gfCNCPoint4[9687] = {X 25.0315, Y 46.1433, Z -5.5000, A 0.000, B 0.000, C 0.000 }
gfCNCPoint4[9688] = {X 23.2598, Y 47.0763, Z -5.5000, A 0.000, B 0.000, C 0.000 }
gfCNCPoint4[9689] = {X 21.4277, Y 47.8844, Z -5.5000, A 0.000, B 0.000, C 0.000 }
gfCNCPoint4[9690] = {X 19.5440, Y 48.5635, Z -5.5000, A 0.000, B 0.000, C 0.000 }
gfCNCPoint4[9691] = {X 19.3880, Y 48.6154, Z -5.5000, A 0.000, B 0.000, C 0.000 }
gfCNCPoint4[9692] = {X 17.4978, Y 49.1350, Z -5.5000, A 0.000, B 0.000, C 0.000 }
gfCNCPoint4[9693] = {X 15.5694, Y 49.4877, Z -5.5000, A 0.000, B 0.000, C 0.000 }
gfCNCPoint4[9694] = {X 13.6177, Y 49.6708, Z -5.5000, A 0.000, B 0.000, C 0.000 }
gfCNCPoint4[9695] = {X 11.6574, Y 49.6828, Z -5.5000, A 0.000, B 0.000, C 0.000 }
gfCNCPoint4[9696] = {X 9.7035, Y 49.5238, Z -5.5000, A 0.000, B 0.000, C 0.000 }
gfCNCPoint4[9697] = {X 7.7709, Y 49.1949, Z -5.5000, A 0.000, B 0.000, C 0.000 }
gfCNCPoint4[9698] = {X 5.9054, Y 48.6841, Z -5.5000, A 0.000, B 0.000, C 0.000 }
gfCNCPoint4[9699] = {X 4.1131, Y 47.9568, Z -5.5000, A 0.000, B 0.000, C 0.000 }
gfCNCPoint4[9700] = {X 2.4191, Y 47.0233, Z -5.5000, A 0.000, B 0.000, C 0.000 }
gfCNCPoint4[9701] = {X 0.8469, Y 45.8966, Z -5.5000, A 0.000, B 0.000, C 0.000 }
gfCNCPoint4[9702] = {X -0.2578, Y 44.9037, Z -5.5000, A 0.000, B 0.000, C 0.000 }
gfCNCPoint4[9703] = {X -1.2389, Y 43.7885, Z -5.5000, A 0.000, B 0.000, C 0.000 }
gfCNCPoint4[9704] = {X -2.0830, Y 42.5663, Z -5.5000, A 0.000, B 0.000, C 0.000 }
gfCNCPoint4[9705] = {X -2.7785, Y 41.2539, Z -5.5000, A 0.000, B 0.000, C 0.000 }
gfCNCPoint4[9706] = {X -3.3159, Y 39.8692, Z -5.5000, A 0.000, B 0.000, C 0.000 }
gfCNCPoint4[9707] = {X -3.5286, Y 39.1333, Z -5.5000, A 0.000, B 0.000, C 0.000 }
gfCNCPoint4[9708] = {X -3.6966, Y 38.3859, Z -5.5000, A 0.000, B 0.000, C 0.000 }
gfCNCPoint4[9709] = {X -4.4555, Y 34.4585, Z -5.5000, A 0.000, B 0.000, C 0.000 }
gfCNCPoint4[9710] = {X -7.9739, Y 34.2502, Z -5.5000, A 0.000, B 0.000, C 0.000 }
gfCNCPoint4[9711] = {X -7.9739, Y 34.2502, Z -2.5000, A 0.000, B 0.000, C 0.000 }
gfCNCPoint4[9712] = {X -7.9739, Y 34.2502, Z 11.0000, A 0.000, B 0.000, C 0.000 }
gfCNCPoint4[9713] = {X 39.8247, Y 26.3830, Z 11.0000, A 0.000, B 0.000, C 0.000 }
gfCNCPoint4[9714] = {X 39.8247, Y 26.3830, Z -2.5000, A 0.000, B 0.000, C 0.000 }
gfCNCPoint4[9715] = {X 39.8247, Y 26.3830, Z -5.5000, A 0.000, B 0.000, C 0.000 }
gfCNCPoint4[9716] = {X 43.6481, Y 27.8072, Z -5.5000, A 0.000, B 0.000, C 0.000 }
gfCNCPoint4[9717] = {X 48.2901, Y 15.3446, Z -5.5000, A 0.000, B 0.000, C 0.000 }
gfCNCPoint4[9718] = {X 47.9079, Y 14.6186, Z -5.5000, A 0.000, B 0.000, C 0.000 }
gfCNCPoint4[9719] = {X 47.6698, Y 13.8334, Z -5.5000, A 0.000, B 0.000, C 0.000 }
gfCNCPoint4[9720] = {X 47.5844, Y 13.0173, Z -5.5000, A 0.000, B 0.000, C 0.000 }
gfCNCPoint4[9721] = {X 47.5842, Y 12.1868, Z -5.5000, A 0.000, B 0.000, C 0.000 }
gfCNCPoint4[9722] = {X 47.6925, Y 11.2255, Z -5.5000, A 0.000, B 0.000, C 0.000 }
gfCNCPoint4[9723] = {X 48.0120, Y 10.3125, Z -5.5000, A 0.000, B 0.000, C 0.000 }
gfCNCPoint4[9724] = {X 48.5267, Y 9.4933, Z -5.5000, A 0.000, B 0.000, C 0.000 }
gfCNCPoint4[9725] = {X 49.2107, Y 8.8093, Z -5.5000, A 0.000, B 0.000, C 0.000 }
gfCNCPoint4[9726] = {X 50.0298, Y 8.2946, Z -5.5000, A 0.000, B 0.000, C 0.000 }
gfCNCPoint4[9727] = {X 50.9429, Y 7.9751, Z -5.5000, A 0.000, B 0.000, C 0.000 }
gfCNCPoint4[9728] = {X 51.9042, Y 7.8668, Z -5.5000, A 0.000, B 0.000, C 0.000 }
gfCNCPoint4[9729] = {X 59.6221, Y 7.8668, Z -5.5000, A 0.000, B 0.000, C 0.000 }
gfCNCPoint4[9730] = {X 60.5834, Y 7.9751, Z -5.5000, A 0.000, B 0.000, C 0.000 }
gfCNCPoint4[9731] = {X 61.4965, Y 8.2946, Z -5.5000, A 0.000, B 0.000, C 0.000 }
gfCNCPoint4[9732] = {X 62.3156, Y 8.8093, Z -5.5000, A 0.000, B 0.000, C 0.000 }
gfCNCPoint4[9733] = {X 62.9996, Y 9.4933, Z -5.5000, A 0.000, B 0.000, C 0.000 }
gfCNCPoint4[9734] = {X 63.5143, Y 10.3124, Z -5.5000, A 0.000, B 0.000, C 0.000 }
gfCNCPoint4[9735] = {X 63.8338, Y 11.2255, Z -5.5000, A 0.000, B 0.000, C 0.000 }
gfCNCPoint4[9736] = {X 63.9421, Y 12.1868, Z -5.5000, A 0.000, B 0.000, C 0.000 }
gfCNCPoint4[9737] = {X 63.9421, Y 12.9782, Z -5.5000, A 0.000, B 0.000, C 0.000 }
gfCNCPoint4[9738] = {X 63.8584, Y 13.8245, Z -5.5000, A 0.000, B 0.000, C 0.000 }
gfCNCPoint4[9739] = {X 63.6104, Y 14.6381, Z -5.5000, A 0.000, B 0.000, C 0.000 }
gfCNCPoint4[9740] = {X 63.2079, Y 15.3874, Z -5.5000, A 0.000, B 0.000, C 0.000 }
gfCNCPoint4[9741] = {X 63.4261, Y 15.9633, Z -5.5000, A 0.000, B 0.000, C 0.000 }
gfCNCPoint4[9742] = {X 66.2401, Y 23.4308, Z -5.5000, A 0.000, B 0.000, C 0.000 }
gfCNCPoint4[9743] = {X 72.2100, Y 39.5004, Z -5.5000, A 0.000, B 0.000, C 0.000 }
gfCNCPoint4[9744] = {X 72.5154, Y 40.2685, Z -5.5000, A 0.000, B 0.000, C 0.000 }
gfCNCPoint4[9745] = {X 73.3597, Y 40.7703, Z -5.5000, A 0.000, B 0.000, C 0.000 }
gfCNCPoint4[9746] = {X 74.0688, Y 41.4499, Z -5.5000, A 0.000, B 0.000, C 0.000 }
gfCNCPoint4[9747] = {X 74.6060, Y 42.2721, Z -5.5000, A 0.000, B 0.000, C 0.000 }
gfCNCPoint4[9748] = {X 74.9437, Y 43.1944, Z -5.5000, A 0.000, B 0.000, C 0.000 }
gfCNCPoint4[9749] = {X 75.0643, Y 44.1692, Z -5.5000, A 0.000, B 0.000, C 0.000 }
gfCNCPoint4[9750] = {X 75.0645, Y 45.0000, Z -5.5000, A 0.000, B 0.000, C 0.000 }
gfCNCPoint4[9751] = {X 74.9561, Y 45.9613, Z -5.5000, A 0.000, B 0.000, C 0.000 }
gfCNCPoint4[9752] = {X 74.6366, Y 46.8744, Z -5.5000, A 0.000, B 0.000, C 0.000 }
gfCNCPoint4[9753] = {X 74.1220, Y 47.6935, Z -5.5000, A 0.000, B 0.000, C 0.000 }
gfCNCPoint4[9754] = {X 73.4379, Y 48.3775, Z -5.5000, A 0.000, B 0.000, C 0.000 }
gfCNCPoint4[9755] = {X 72.6188, Y 48.8922, Z -5.5000, A 0.000, B 0.000, C 0.000 }
gfCNCPoint4[9756] = {X 71.7057, Y 49.2117, Z -5.5000, A 0.000, B 0.000, C 0.000 }
gfCNCPoint4[9757] = {X 70.7445, Y 49.3200, Z -5.5000, A 0.000, B 0.000, C 0.000 }
gfCNCPoint4[9758] = {X 64.1851, Y 49.3200, Z -5.5000, A 0.000, B 0.000, C 0.000 }
gfCNCPoint4[9759] = {X 63.2238, Y 49.2117, Z -5.5000, A 0.000, B 0.000, C 0.000 }
gfCNCPoint4[9760] = {X 62.3108, Y 48.8922, Z -5.5000, A 0.000, B 0.000, C 0.000 }
gfCNCPoint4[9761] = {X 61.4917, Y 48.3775, Z -5.5000, A 0.000, B 0.000, C 0.000 }
gfCNCPoint4[9762] = {X 60.8076, Y 47.6935, Z -5.5000, A 0.000, B 0.000, C 0.000 }
gfCNCPoint4[9763] = {X 60.2929, Y 46.8744, Z -5.5000, A 0.000, B 0.000, C 0.000 }
gfCNCPoint4[9764] = {X 59.9734, Y 45.9613, Z -5.5000, A 0.000, B 0.000, C 0.000 }
gfCNCPoint4[9765] = {X 59.8651, Y 45.0000, Z -5.5000, A 0.000, B 0.000, C 0.000 }
gfCNCPoint4[9766] = {X 59.8651, Y 44.2085, Z -5.5000, A 0.000, B 0.000, C 0.000 }
gfCNCPoint4[9767] = {X 59.9518, Y 43.3502, Z -5.5000, A 0.000, B 0.000, C 0.000 }
gfCNCPoint4[9768] = {X 60.2072, Y 42.5262, Z -5.5000, A 0.000, B 0.000, C 0.000 }
gfCNCPoint4[9769] = {X 60.6213, Y 41.7694, Z -5.5000, A 0.000, B 0.000, C 0.000 }
gfCNCPoint4[9770] = {X 60.0068, Y 40.0892, Z -5.5000, A 0.000, B 0.000, C 0.000 }
gfCNCPoint4[9771] = {X 52.0776, Y 40.0892, Z -5.5000, A 0.000, B 0.000, C 0.000 }
gfCNCPoint4[9772] = {X 51.3347, Y 42.0851, Z -5.5000, A 0.000, B 0.000, C 0.000 }
gfCNCPoint4[9773] = {X 51.3378, Y 42.0902, Z -5.5000, A 0.000, B 0.000, C 0.000 }
gfCNCPoint4[9774] = {X 51.6390, Y 42.7496, Z -5.5000, A 0.000, B 0.000, C 0.000 }
gfCNCPoint4[9775] = {X 51.8258, Y 43.4501, Z -5.5000, A 0.000, B 0.000, C 0.000 }
gfCNCPoint4[9776] = {X 51.8928, Y 44.1720, Z -5.5000, A 0.000, B 0.000, C 0.000 }
gfCNCPoint4[9777] = {X 51.8929, Y 45.0000, Z -5.5000, A 0.000, B 0.000, C 0.000 }
gfCNCPoint4[9778] = {X 51.7846, Y 45.9613, Z -5.5000, A 0.000, B 0.000, C 0.000 }
gfCNCPoint4[9779] = {X 51.4651, Y 46.8744, Z -5.5000, A 0.000, B 0.000, C 0.000 }
gfCNCPoint4[9780] = {X 50.9504, Y 47.6935, Z -5.5000, A 0.000, B 0.000, C 0.000 }
gfCNCPoint4[9781] = {X 50.2664, Y 48.3775, Z -5.5000, A 0.000, B 0.000, C 0.000 }
gfCNCPoint4[9782] = {X 49.4473, Y 48.8922, Z -5.5000, A 0.000, B 0.000, C 0.000 }
gfCNCPoint4[9783] = {X 48.5342, Y 49.2117, Z -5.5000, A 0.000, B 0.000, C 0.000 }
gfCNCPoint4[9784] = {X 47.5729, Y 49.3200, Z -5.5000, A 0.000, B 0.000, C 0.000 }
gfCNCPoint4[9785] = {X 40.6393, Y 49.3200, Z -5.5000, A 0.000, B 0.000, C 0.000 }
gfCNCPoint4[9786] = {X 39.6780, Y 49.2117, Z -5.5000, A 0.000, B 0.000, C 0.000 }
gfCNCPoint4[9787] = {X 38.7649, Y 48.8922, Z -5.5000, A 0.000, B 0.000, C 0.000 }
gfCNCPoint4[9788] = {X 37.9458, Y 48.3775, Z -5.5000, A 0.000, B 0.000, C 0.000 }
gfCNCPoint4[9789] = {X 37.2618, Y 47.6935, Z -5.5000, A 0.000, B 0.000, C 0.000 }
gfCNCPoint4[9790] = {X 36.7471, Y 46.8744, Z -5.5000, A 0.000, B 0.000, C 0.000 }
gfCNCPoint4[9791] = {X 36.4276, Y 45.9613, Z -5.5000, A 0.000, B 0.000, C 0.000 }
gfCNCPoint4[9792] = {X 36.3193, Y 45.0000, Z -5.5000, A 0.000, B 0.000, C 0.000 }
gfCNCPoint4[9793] = {X 36.3193, Y 44.2086, Z -5.5000, A 0.000, B 0.000, C 0.000 }
gfCNCPoint4[9794] = {X 36.4360, Y 43.2115, Z -5.5000, A 0.000, B 0.000, C 0.000 }
gfCNCPoint4[9795] = {X 36.7796, Y 42.2683, Z -5.5000, A 0.000, B 0.000, C 0.000 }
gfCNCPoint4[9796] = {X 37.3317, Y 41.4299, Z -5.5000, A 0.000, B 0.000, C 0.000 }
gfCNCPoint4[9797] = {X 38.0624, Y 40.7415, Z -5.5000, A 0.000, B 0.000, C 0.000 }
gfCNCPoint4[9798] = {X 38.9322, Y 40.2404, Z -5.5000, A 0.000, B 0.000, C 0.000 }
gfCNCPoint4[9799] = {X 39.5233, Y 38.8448, Z -5.5000, A 0.000, B 0.000, C 0.000 }
gfCNCPoint4[9800] = {X 40.0641, Y 37.4291, Z -5.5000, A 0.000, B 0.000, C 0.000 }
gfCNCPoint4[9801] = {X 43.6481, Y 27.8072, Z -5.5000, A 0.000, B 0.000, C 0.000 }
gfCNCPoint4[9802] = {X 39.8997, Y 26.4110, Z -5.5000, A 0.000, B 0.000, C 0.000 }
gfCNCPoint4[9803] = {X 43.7231, Y 27.8351, Z -5.5000, A 0.000, B 0.000, C 0.000 }
gfCNCPoint4[9804] = {X 48.3793, Y 15.3344, Z -5.5000, A 0.000, B 0.000, C 0.000 }
gfCNCPoint4[9805] = {X 47.9922, Y 14.6130, Z -5.5000, A 0.000, B 0.000, C 0.000 }
gfCNCPoint4[9806] = {X 47.7508, Y 13.8307, Z -5.5000, A 0.000, B 0.000, C 0.000 }
gfCNCPoint4[9807] = {X 47.6644, Y 13.0166, Z -5.5000, A 0.000, B 0.000, C 0.000 }
gfCNCPoint4[9808] = {X 47.6642, Y 12.1868, Z -5.5000, A 0.000, B 0.000, C 0.000 }
gfCNCPoint4[9809] = {X 47.7705, Y 11.2433, Z -5.5000, A 0.000, B 0.000, C 0.000 }
gfCNCPoint4[9810] = {X 48.0841, Y 10.3472, Z -5.5000, A 0.000, B 0.000, C 0.000 }
gfCNCPoint4[9811] = {X 48.5893, Y 9.5432, Z -5.5000, A 0.000, B 0.000, C 0.000 }
gfCNCPoint4[9812] = {X 49.2606, Y 8.8719, Z -5.5000, A 0.000, B 0.000, C 0.000 }
gfCNCPoint4[9813] = {X 50.0646, Y 8.3667, Z -5.5000, A 0.000, B 0.000, C 0.000 }
gfCNCPoint4[9814] = {X 50.9607, Y 8.0531, Z -5.5000, A 0.000, B 0.000, C 0.000 }
gfCNCPoint4[9815] = {X 51.9042, Y 7.9468, Z -5.5000, A 0.000, B 0.000, C 0.000 }
gfCNCPoint4[9816] = {X 59.6221, Y 7.9468, Z -5.5000, A 0.000, B 0.000, C 0.000 }
gfCNCPoint4[9817] = {X 60.5656, Y 8.0531, Z -5.5000, A 0.000, B 0.000, C 0.000 }
gfCNCPoint4[9818] = {X 61.4618, Y 8.3667, Z -5.5000, A 0.000, B 0.000, C 0.000 }
gfCNCPoint4[9819] = {X 62.2657, Y 8.8718, Z -5.5000, A 0.000, B 0.000, C 0.000 }
gfCNCPoint4[9820] = {X 62.9371, Y 9.5432, Z -5.5000, A 0.000, B 0.000, C 0.000 }
gfCNCPoint4[9821] = {X 63.4422, Y 10.3471, Z -5.5000, A 0.000, B 0.000, C 0.000 }
gfCNCPoint4[9822] = {X 63.7558, Y 11.2433, Z -5.5000, A 0.000, B 0.000, C 0.000 }
gfCNCPoint4[9823] = {X 63.8621, Y 12.1868, Z -5.5000, A 0.000, B 0.000, C 0.000 }
gfCNCPoint4[9824] = {X 63.8621, Y 12.9782, Z -5.5000, A 0.000, B 0.000, C 0.000 }
gfCNCPoint4[9825] = {X 63.7772, Y 13.8223, Z -5.5000, A 0.000, B 0.000, C 0.000 }
gfCNCPoint4[9826] = {X 63.5259, Y 14.6327, Z -5.5000, A 0.000, B 0.000, C 0.000 }
gfCNCPoint4[9827] = {X 63.1183, Y 15.3768, Z -5.5000, A 0.000, B 0.000, C 0.000 }
gfCNCPoint4[9828] = {X 63.3513, Y 15.9916, Z -5.5000, A 0.000, B 0.000, C 0.000 }
gfCNCPoint4[9829] = {X 66.1652, Y 23.4588, Z -5.5000, A 0.000, B 0.000, C 0.000 }
gfCNCPoint4[9830] = {X 72.1353, Y 39.5291, Z -5.5000, A 0.000, B 0.000, C 0.000 }
gfCNCPoint4[9831] = {X 72.4531, Y 40.3283, Z -5.5000, A 0.000, B 0.000, C 0.000 }
gfCNCPoint4[9832] = {X 73.2906, Y 40.8184, Z -5.5000, A 0.000, B 0.000, C 0.000 }
gfCNCPoint4[9833] = {X 73.9948, Y 41.4861, Z -5.5000, A 0.000, B 0.000, C 0.000 }
gfCNCPoint4[9834] = {X 74.5287, Y 42.2964, Z -5.5000, A 0.000, B 0.000, C 0.000 }
gfCNCPoint4[9835] = {X 74.8644, Y 43.2069, Z -5.5000, A 0.000, B 0.000, C 0.000 }
gfCNCPoint4[9836] = {X 74.9843, Y 44.1699, Z -5.5000, A 0.000, B 0.000, C 0.000 }
gfCNCPoint4[9837] = {X 74.9845, Y 45.0000, Z -5.5000, A 0.000, B 0.000, C 0.000 }
gfCNCPoint4[9838] = {X 74.8782, Y 45.9435, Z -5.5000, A 0.000, B 0.000, C 0.000 }
gfCNCPoint4[9839] = {X 74.5646, Y 46.8397, Z -5.5000, A 0.000, B 0.000, C 0.000 }
gfCNCPoint4[9840] = {X 74.0594, Y 47.6436, Z -5.5000, A 0.000, B 0.000, C 0.000 }
gfCNCPoint4[9841] = {X 73.3881, Y 48.3150, Z -5.5000, A 0.000, B 0.000, C 0.000 }
gfCNCPoint4[9842] = {X 72.5841, Y 48.8201, Z -5.5000, A 0.000, B 0.000, C 0.000 }
gfCNCPoint4[9843] = {X 71.6879, Y 49.1337, Z -5.5000, A 0.000, B 0.000, C 0.000 }
gfCNCPoint4[9844] = {X 70.7445, Y 49.2400, Z -5.5000, A 0.000, B 0.000, C 0.000 }
gfCNCPoint4[9845] = {X 64.1851, Y 49.2400, Z -5.5000, A 0.000, B 0.000, C 0.000 }
gfCNCPoint4[9846] = {X 63.2416, Y 49.1337, Z -5.5000, A 0.000, B 0.000, C 0.000 }
gfCNCPoint4[9847] = {X 62.3455, Y 48.8201, Z -5.5000, A 0.000, B 0.000, C 0.000 }
gfCNCPoint4[9848] = {X 61.5415, Y 48.3150, Z -5.5000, A 0.000, B 0.000, C 0.000 }
gfCNCPoint4[9849] = {X 60.8702, Y 47.6436, Z -5.5000, A 0.000, B 0.000, C 0.000 }
gfCNCPoint4[9850] = {X 60.3650, Y 46.8397, Z -5.5000, A 0.000, B 0.000, C 0.000 }
gfCNCPoint4[9851] = {X 60.0514, Y 45.9435, Z -5.5000, A 0.000, B 0.000, C 0.000 }
gfCNCPoint4[9852] = {X 59.9451, Y 45.0000, Z -5.5000, A 0.000, B 0.000, C 0.000 }
gfCNCPoint4[9853] = {X 59.9451, Y 44.2085, Z -5.5000, A 0.000, B 0.000, C 0.000 }
gfCNCPoint4[9854] = {X 60.0329, Y 43.3527, Z -5.5000, A 0.000, B 0.000, C 0.000 }
gfCNCPoint4[9855] = {X 60.2917, Y 42.5322, Z -5.5000, A 0.000, B 0.000, C 0.000 }
gfCNCPoint4[9856] = {X 60.7107, Y 41.7808, Z -5.5000, A 0.000, B 0.000, C 0.000 }
gfCNCPoint4[9857] = {X 60.0627, Y 40.0092, Z -5.5000, A 0.000, B 0.000, C 0.000 }
gfCNCPoint4[9858] = {X 52.0220, Y 40.0092, Z -5.5000, A 0.000, B 0.000, C 0.000 }
gfCNCPoint4[9859] = {X 51.2464, Y 42.0932, Z -5.5000, A 0.000, B 0.000, C 0.000 }
gfCNCPoint4[9860] = {X 51.2685, Y 42.1303, Z -5.5000, A 0.000, B 0.000, C 0.000 }
gfCNCPoint4[9861] = {X 51.5640, Y 42.7773, Z -5.5000, A 0.000, B 0.000, C 0.000 }
gfCNCPoint4[9862] = {X 51.7471, Y 43.4645, Z -5.5000, A 0.000, B 0.000, C 0.000 }
gfCNCPoint4[9863] = {X 51.8128, Y 44.1726, Z -5.5000, A 0.000, B 0.000, C 0.000 }
gfCNCPoint4[9864] = {X 51.8129, Y 45.0000, Z -5.5000, A 0.000, B 0.000, C 0.000 }
gfCNCPoint4[9865] = {X 51.7066, Y 45.9435, Z -5.5000, A 0.000, B 0.000, C 0.000 }
gfCNCPoint4[9866] = {X 51.3930, Y 46.8397, Z -5.5000, A 0.000, B 0.000, C 0.000 }
gfCNCPoint4[9867] = {X 50.8879, Y 47.6436, Z -5.5000, A 0.000, B 0.000, C 0.000 }
gfCNCPoint4[9868] = {X 50.2165, Y 48.3150, Z -5.5000, A 0.000, B 0.000, C 0.000 }
gfCNCPoint4[9869] = {X 49.4126, Y 48.8201, Z -5.5000, A 0.000, B 0.000, C 0.000 }
gfCNCPoint4[9870] = {X 48.5164, Y 49.1337, Z -5.5000, A 0.000, B 0.000, C 0.000 }
gfCNCPoint4[9871] = {X 47.5729, Y 49.2400, Z -5.5000, A 0.000, B 0.000, C 0.000 }
gfCNCPoint4[9872] = {X 40.6393, Y 49.2400, Z -5.5000, A 0.000, B 0.000, C 0.000 }
gfCNCPoint4[9873] = {X 39.6958, Y 49.1337, Z -5.5000, A 0.000, B 0.000, C 0.000 }
gfCNCPoint4[9874] = {X 38.7996, Y 48.8201, Z -5.5000, A 0.000, B 0.000, C 0.000 }
gfCNCPoint4[9875] = {X 37.9957, Y 48.3150, Z -5.5000, A 0.000, B 0.000, C 0.000 }
gfCNCPoint4[9876] = {X 37.3243, Y 47.6436, Z -5.5000, A 0.000, B 0.000, C 0.000 }
gfCNCPoint4[9877] = {X 36.8192, Y 46.8397, Z -5.5000, A 0.000, B 0.000, C 0.000 }
gfCNCPoint4[9878] = {X 36.5056, Y 45.9435, Z -5.5000, A 0.000, B 0.000, C 0.000 }
gfCNCPoint4[9879] = {X 36.3993, Y 45.0000, Z -5.5000, A 0.000, B 0.000, C 0.000 }
gfCNCPoint4[9880] = {X 36.3993, Y 44.2086, Z -5.5000, A 0.000, B 0.000, C 0.000 }
gfCNCPoint4[9881] = {X 36.5153, Y 43.2240, Z -5.5000, A 0.000, B 0.000, C 0.000 }
gfCNCPoint4[9882] = {X 36.8567, Y 42.2931, Z -5.5000, A 0.000, B 0.000, C 0.000 }
gfCNCPoint4[9883] = {X 37.4050, Y 41.4671, Z -5.5000, A 0.000, B 0.000, C 0.000 }
gfCNCPoint4[9884] = {X 38.1301, Y 40.7909, Z -5.5000, A 0.000, B 0.000, C 0.000 }
gfCNCPoint4[9885] = {X 38.9925, Y 40.3017, Z -5.5000, A 0.000, B 0.000, C 0.000 }
gfCNCPoint4[9886] = {X 39.5916, Y 38.8893, Z -5.5000, A 0.000, B 0.000, C 0.000 }
gfCNCPoint4[9887] = {X 40.1394, Y 37.4563, Z -5.5000, A 0.000, B 0.000, C 0.000 }
gfCNCPoint4[9888] = {X 43.7231, Y 27.8351, Z -5.5000, A 0.000, B 0.000, C 0.000 }
gfCNCPoint4[9889] = {X 39.9746, Y 26.4389, Z -5.5000, A 0.000, B 0.000, C 0.000 }
gfCNCPoint4[9890] = {X 43.7980, Y 27.8630, Z -5.5000, A 0.000, B 0.000, C 0.000 }
gfCNCPoint4[9891] = {X 48.4687, Y 15.3238, Z -5.5000, A 0.000, B 0.000, C 0.000 }
gfCNCPoint4[9892] = {X 48.0765, Y 14.6072, Z -5.5000, A 0.000, B 0.000, C 0.000 }
gfCNCPoint4[9893] = {X 47.8320, Y 13.8279, Z -5.5000, A 0.000, B 0.000, C 0.000 }
gfCNCPoint4[9894] = {X 47.7444, Y 13.0158, Z -5.5000, A 0.000, B 0.000, C 0.000 }
gfCNCPoint4[9895] = {X 47.7442, Y 12.1868, Z -5.5000, A 0.000, B 0.000, C 0.000 }
gfCNCPoint4[9896] = {X 47.8485, Y 11.2611, Z -5.5000, A 0.000, B 0.000, C 0.000 }
gfCNCPoint4[9897] = {X 48.1562, Y 10.3819, Z -5.5000, A 0.000, B 0.000, C 0.000 }
gfCNCPoint4[9898] = {X 48.6518, Y 9.5931, Z -5.5000, A 0.000, B 0.000, C 0.000 }
gfCNCPoint4[9899] = {X 49.3105, Y 8.9344, Z -5.5000, A 0.000, B 0.000, C 0.000 }
gfCNCPoint4[9900] = {X 50.0993, Y 8.4388, Z -5.5000, A 0.000, B 0.000, C 0.000 }
gfCNCPoint4[9901] = {X 50.9785, Y 8.1311, Z -5.5000, A 0.000, B 0.000, C 0.000 }
gfCNCPoint4[9902] = {X 51.9042, Y 8.0268, Z -5.5000, A 0.000, B 0.000, C 0.000 }
gfCNCPoint4[9903] = {X 59.6221, Y 8.0268, Z -5.5000, A 0.000, B 0.000, C 0.000 }
gfCNCPoint4[9904] = {X 60.5478, Y 8.1311, Z -5.5000, A 0.000, B 0.000, C 0.000 }
gfCNCPoint4[9905] = {X 61.4271, Y 8.4388, Z -5.5000, A 0.000, B 0.000, C 0.000 }
gfCNCPoint4[9906] = {X 62.2158, Y 8.9344, Z -5.5000, A 0.000, B 0.000, C 0.000 }
gfCNCPoint4[9907] = {X 62.8745, Y 9.5931, Z -5.5000, A 0.000, B 0.000, C 0.000 }
gfCNCPoint4[9908] = {X 63.3702, Y 10.3819, Z -5.5000, A 0.000, B 0.000, C 0.000 }
gfCNCPoint4[9909] = {X 63.6778, Y 11.2611, Z -5.5000, A 0.000, B 0.000, C 0.000 }
gfCNCPoint4[9910] = {X 63.7821, Y 12.1868, Z -5.5000, A 0.000, B 0.000, C 0.000 }
gfCNCPoint4[9911] = {X 63.7821, Y 12.9782, Z -5.5000, A 0.000, B 0.000, C 0.000 }
gfCNCPoint4[9912] = {X 63.6960, Y 13.8200, Z -5.5000, A 0.000, B 0.000, C 0.000 }
gfCNCPoint4[9913] = {X 63.4413, Y 14.6270, Z -5.5000, A 0.000, B 0.000, C 0.000 }
gfCNCPoint4[9914] = {X 63.0286, Y 15.3658, Z -5.5000, A 0.000, B 0.000, C 0.000 }
gfCNCPoint4[9915] = {X 63.2765, Y 16.0199, Z -5.5000, A 0.000, B 0.000, C 0.000 }
gfCNCPoint4[9916] = {X 66.0903, Y 23.4869, Z -5.5000, A 0.000, B 0.000, C 0.000 }
gfCNCPoint4[9917] = {X 72.0607, Y 39.5578, Z -5.5000, A 0.000, B 0.000, C 0.000 }
gfCNCPoint4[9918] = {X 72.3909, Y 40.3885, Z -5.5000, A 0.000, B 0.000, C 0.000 }
gfCNCPoint4[9919] = {X 73.2216, Y 40.8668, Z -5.5000, A 0.000, B 0.000, C 0.000 }
gfCNCPoint4[9920] = {X 73.9208, Y 41.5225, Z -5.5000, A 0.000, B 0.000, C 0.000 }
gfCNCPoint4[9921] = {X 74.4514, Y 42.3209, Z -5.5000, A 0.000, B 0.000, C 0.000 }
gfCNCPoint4[9922] = {X 74.7851, Y 43.2195, Z -5.5000, A 0.000, B 0.000, C 0.000 }
gfCNCPoint4[9923] = {X 74.9043, Y 44.1706, Z -5.5000, A 0.000, B 0.000, C 0.000 }
gfCNCPoint4[9924] = {X 74.9045, Y 45.0000, Z -5.5000, A 0.000, B 0.000, C 0.000 }
gfCNCPoint4[9925] = {X 74.8002, Y 45.9257, Z -5.5000, A 0.000, B 0.000, C 0.000 }
gfCNCPoint4[9926] = {X 74.4925, Y 46.8050, Z -5.5000, A 0.000, B 0.000, C 0.000 }
gfCNCPoint4[9927] = {X 73.9969, Y 47.5937, Z -5.5000, A 0.000, B 0.000, C 0.000 }
gfCNCPoint4[9928] = {X 73.3382, Y 48.2524, Z -5.5000, A 0.000, B 0.000, C 0.000 }
gfCNCPoint4[9929] = {X 72.5494, Y 48.7480, Z -5.5000, A 0.000, B 0.000, C 0.000 }
gfCNCPoint4[9930] = {X 71.6701, Y 49.0557, Z -5.5000, A 0.000, B 0.000, C 0.000 }
gfCNCPoint4[9931] = {X 70.7445, Y 49.1600, Z -5.5000, A 0.000, B 0.000, C 0.000 }
gfCNCPoint4[9932] = {X 64.1851, Y 49.1600, Z -5.5000, A 0.000, B 0.000, C 0.000 }
gfCNCPoint4[9933] = {X 63.2594, Y 49.0557, Z -5.5000, A 0.000, B 0.000, C 0.000 }
gfCNCPoint4[9934] = {X 62.3802, Y 48.7480, Z -5.5000, A 0.000, B 0.000, C 0.000 }
gfCNCPoint4[9935] = {X 61.5914, Y 48.2524, Z -5.5000, A 0.000, B 0.000, C 0.000 }
gfCNCPoint4[9936] = {X 60.9327, Y 47.5937, Z -5.5000, A 0.000, B 0.000, C 0.000 }
gfCNCPoint4[9937] = {X 60.4371, Y 46.8050, Z -5.5000, A 0.000, B 0.000, C 0.000 }
gfCNCPoint4[9938] = {X 60.1294, Y 45.9257, Z -5.5000, A 0.000, B 0.000, C 0.000 }
gfCNCPoint4[9939] = {X 60.0251, Y 45.0000, Z -5.5000, A 0.000, B 0.000, C 0.000 }
gfCNCPoint4[9940] = {X 60.0251, Y 44.2086, Z -5.5000, A 0.000, B 0.000, C 0.000 }
gfCNCPoint4[9941] = {X 60.1141, Y 43.3553, Z -5.5000, A 0.000, B 0.000, C 0.000 }
gfCNCPoint4[9942] = {X 60.3762, Y 42.5385, Z -5.5000, A 0.000, B 0.000, C 0.000 }
gfCNCPoint4[9943] = {X 60.8002, Y 41.7927, Z -5.5000, A 0.000, B 0.000, C 0.000 }
gfCNCPoint4[9944] = {X 60.1186, Y 39.9292, Z -5.5000, A 0.000, B 0.000, C 0.000 }
gfCNCPoint4[9945] = {X 51.9665, Y 39.9292, Z -5.5000, A 0.000, B 0.000, C 0.000 }
gfCNCPoint4[9946] = {X 51.1580, Y 42.1013, Z -5.5000, A 0.000, B 0.000, C 0.000 }
gfCNCPoint4[9947] = {X 51.1993, Y 42.1704, Z -5.5000, A 0.000, B 0.000, C 0.000 }
gfCNCPoint4[9948] = {X 51.4889, Y 42.8049, Z -5.5000, A 0.000, B 0.000, C 0.000 }
gfCNCPoint4[9949] = {X 51.6684, Y 43.4789, Z -5.5000, A 0.000, B 0.000, C 0.000 }
gfCNCPoint4[9950] = {X 51.7328, Y 44.1733, Z -5.5000, A 0.000, B 0.000, C 0.000 }
gfCNCPoint4[9951] = {X 51.7329, Y 45.0000, Z -5.5000, A 0.000, B 0.000, C 0.000 }
gfCNCPoint4[9952] = {X 51.6286, Y 45.9257, Z -5.5000, A 0.000, B 0.000, C 0.000 }
gfCNCPoint4[9953] = {X 51.3210, Y 46.8050, Z -5.5000, A 0.000, B 0.000, C 0.000 }
gfCNCPoint4[9954] = {X 50.8253, Y 47.5937, Z -5.5000, A 0.000, B 0.000, C 0.000 }
gfCNCPoint4[9955] = {X 50.1666, Y 48.2524, Z -5.5000, A 0.000, B 0.000, C 0.000 }
gfCNCPoint4[9956] = {X 49.3779, Y 48.7480, Z -5.5000, A 0.000, B 0.000, C 0.000 }
gfCNCPoint4[9957] = {X 48.4986, Y 49.0557, Z -5.5000, A 0.000, B 0.000, C 0.000 }
gfCNCPoint4[9958] = {X 47.5729, Y 49.1600, Z -5.5000, A 0.000, B 0.000, C 0.000 }
gfCNCPoint4[9959] = {X 40.6393, Y 49.1600, Z -5.5000, A 0.000, B 0.000, C 0.000 }
gfCNCPoint4[9960] = {X 39.7136, Y 49.0557, Z -5.5000, A 0.000, B 0.000, C 0.000 }
gfCNCPoint4[9961] = {X 38.8343, Y 48.7480, Z -5.5000, A 0.000, B 0.000, C 0.000 }
gfCNCPoint4[9962] = {X 38.0456, Y 48.2524, Z -5.5000, A 0.000, B 0.000, C 0.000 }
gfCNCPoint4[9963] = {X 37.3869, Y 47.5937, Z -5.5000, A 0.000, B 0.000, C 0.000 }
gfCNCPoint4[9964] = {X 36.8913, Y 46.8050, Z -5.5000, A 0.000, B 0.000, C 0.000 }
gfCNCPoint4[9965] = {X 36.5836, Y 45.9257, Z -5.5000, A 0.000, B 0.000, C 0.000 }
gfCNCPoint4[9966] = {X 36.4793, Y 45.0000, Z -5.5000, A 0.000, B 0.000, C 0.000 }
gfCNCPoint4[9967] = {X 36.4793, Y 44.2086, Z -5.5000, A 0.000, B 0.000, C 0.000 }
gfCNCPoint4[9968] = {X 36.5945, Y 43.2364, Z -5.5000, A 0.000, B 0.000, C 0.000 }
gfCNCPoint4[9969] = {X 36.9338, Y 42.3181, Z -5.5000, A 0.000, B 0.000, C 0.000 }
gfCNCPoint4[9970] = {X 37.4783, Y 41.5044, Z -5.5000, A 0.000, B 0.000, C 0.000 }
gfCNCPoint4[9971] = {X 38.1978, Y 40.8406, Z -5.5000, A 0.000, B 0.000, C 0.000 }
gfCNCPoint4[9972] = {X 39.0526, Y 40.3633, Z -5.5000, A 0.000, B 0.000, C 0.000 }
gfCNCPoint4[9973] = {X 39.6598, Y 38.9340, Z -5.5000, A 0.000, B 0.000, C 0.000 }
gfCNCPoint4[9974] = {X 40.2146, Y 37.4835, Z -5.5000, A 0.000, B 0.000, C 0.000 }
gfCNCPoint4[9975] = {X 43.7980, Y 27.8630, Z -5.5000, A 0.000, B 0.000, C 0.000 }
gfCNCPoint4[9976] = {X 40.0496, Y 26.4668, Z -5.5000, A 0.000, B 0.000, C 0.000 }
gfCNCPoint4[9977] = {X 43.8730, Y 27.8909, Z -5.5000, A 0.000, B 0.000, C 0.000 }
gfCNCPoint4[9978] = {X 48.5582, Y 15.3126, Z -5.5000, A 0.000, B 0.000, C 0.000 }
gfCNCPoint4[9979] = {X 48.1610, Y 14.6012, Z -5.5000, A 0.000, B 0.000, C 0.000 }
gfCNCPoint4[9980] = {X 47.9131, Y 13.8250, Z -5.5000, A 0.000, B 0.000, C 0.000 }
gfCNCPoint4[9981] = {X 47.8244, Y 13.0151, Z -5.5000, A 0.000, B 0.000, C 0.000 }
gfCNCPoint4[9982] = {X 47.8242, Y 12.1868, Z -5.5000, A 0.000, B 0.000, C 0.000 }
gfCNCPoint4[9983] = {X 47.9265, Y 11.2789, Z -5.5000, A 0.000, B 0.000, C 0.000 }
gfCNCPoint4[9984] = {X 48.2283, Y 10.4166, Z -5.5000, A 0.000, B 0.000, C 0.000 }
gfCNCPoint4[9985] = {X 48.7144, Y 9.6430, Z -5.5000, A 0.000, B 0.000, C 0.000 }
gfCNCPoint4[9986] = {X 49.3604, Y 8.9969, Z -5.5000, A 0.000, B 0.000, C 0.000 }
gfCNCPoint4[9987] = {X 50.1340, Y 8.5109, Z -5.5000, A 0.000, B 0.000, C 0.000 }
gfCNCPoint4[9988] = {X 50.9963, Y 8.2091, Z -5.5000, A 0.000, B 0.000, C 0.000 }
gfCNCPoint4[9989] = {X 51.9042, Y 8.1068, Z -5.5000, A 0.000, B 0.000, C 0.000 }
gfCNCPoint4[9990] = {X 59.6221, Y 8.1068, Z -5.5000, A 0.000, B 0.000, C 0.000 }
gfCNCPoint4[9991] = {X 60.5300, Y 8.2091, Z -5.5000, A 0.000, B 0.000, C 0.000 }
gfCNCPoint4[9992] = {X 61.3924, Y 8.5109, Z -5.5000, A 0.000, B 0.000, C 0.000 }
gfCNCPoint4[9993] = {X 62.1660, Y 8.9969, Z -5.5000, A 0.000, B 0.000, C 0.000 }
gfCNCPoint4[9994] = {X 62.8120, Y 9.6430, Z -5.5000, A 0.000, B 0.000, C 0.000 }
gfCNCPoint4[9995] = {X 63.2981, Y 10.4166, Z -5.5000, A 0.000, B 0.000, C 0.000 }
gfCNCPoint4[9996] = {X 63.5998, Y 11.2789, Z -5.5000, A 0.000, B 0.000, C 0.000 }
gfCNCPoint4[9997] = {X 63.7021, Y 12.1868, Z -5.5000, A 0.000, B 0.000, C 0.000 }
gfCNCPoint4[9998] = {X 63.7021, Y 12.9782, Z -5.5000, A 0.000, B 0.000, C 0.000 }
gfCNCPoint4[9999] = {X 63.6148, Y 13.8176, Z -5.5000, A 0.000, B 0.000, C 0.000 }
gfCNCPoint4[10000] = {X 63.3566, Y 14.6211, Z -5.5000, A 0.000, B 0.000, C 0.000 }
gfCNCPoint4[10001] = {X 62.9387, Y 15.3543, Z -5.5000, A 0.000, B 0.000, C 0.000 }
gfCNCPoint4[10002] = {X 63.2016, Y 16.0481, Z -5.5000, A 0.000, B 0.000, C 0.000 }
gfCNCPoint4[10003] = {X 66.0153, Y 23.5149, Z -5.5000, A 0.000, B 0.000, C 0.000 }
gfCNCPoint4[10004] = {X 71.9860, Y 39.5865, Z -5.5000, A 0.000, B 0.000, C 0.000 }
gfCNCPoint4[10005] = {X 72.3289, Y 40.4490, Z -5.5000, A 0.000, B 0.000, C 0.000 }
gfCNCPoint4[10006] = {X 73.1527, Y 40.9154, Z -5.5000, A 0.000, B 0.000, C 0.000 }
gfCNCPoint4[10007] = {X 73.8469, Y 41.5591, Z -5.5000, A 0.000, B 0.000, C 0.000 }
gfCNCPoint4[10008] = {X 74.3741, Y 42.3454, Z -5.5000, A 0.000, B 0.000, C 0.000 }
gfCNCPoint4[10009] = {X 74.7058, Y 43.2321, Z -5.5000, A 0.000, B 0.000, C 0.000 }
gfCNCPoint4[10010] = {X 74.8243, Y 44.1714, Z -5.5000, A 0.000, B 0.000, C 0.000 }
gfCNCPoint4[10011] = {X 74.8245, Y 45.0000, Z -5.5000, A 0.000, B 0.000, C 0.000 }
gfCNCPoint4[10012] = {X 74.7222, Y 45.9079, Z -5.5000, A 0.000, B 0.000, C 0.000 }
gfCNCPoint4[10013] = {X 74.4204, Y 46.7702, Z -5.5000, A 0.000, B 0.000, C 0.000 }
gfCNCPoint4[10014] = {X 73.9343, Y 47.5438, Z -5.5000, A 0.000, B 0.000, C 0.000 }
gfCNCPoint4[10015] = {X 73.2883, Y 48.1899, Z -5.5000, A 0.000, B 0.000, C 0.000 }
gfCNCPoint4[10016] = {X 72.5147, Y 48.6760, Z -5.5000, A 0.000, B 0.000, C 0.000 }
gfCNCPoint4[10017] = {X 71.6523, Y 48.9777, Z -5.5000, A 0.000, B 0.000, C 0.000 }
gfCNCPoint4[10018] = {X 70.7445, Y 49.0800, Z -5.5000, A 0.000, B 0.000, C 0.000 }
gfCNCPoint4[10019] = {X 64.1851, Y 49.0800, Z -5.5000, A 0.000, B 0.000, C 0.000 }
gfCNCPoint4[10020] = {X 63.2772, Y 48.9777, Z -5.5000, A 0.000, B 0.000, C 0.000 }
gfCNCPoint4[10021] = {X 62.4149, Y 48.6760, Z -5.5000, A 0.000, B 0.000, C 0.000 }
gfCNCPoint4[10022] = {X 61.6413, Y 48.1899, Z -5.5000, A 0.000, B 0.000, C 0.000 }
gfCNCPoint4[10023] = {X 60.9953, Y 47.5438, Z -5.5000, A 0.000, B 0.000, C 0.000 }
gfCNCPoint4[10024] = {X 60.5092, Y 46.7702, Z -5.5000, A 0.000, B 0.000, C 0.000 }
gfCNCPoint4[10025] = {X 60.2074, Y 45.9079, Z -5.5000, A 0.000, B 0.000, C 0.000 }
gfCNCPoint4[10026] = {X 60.1051, Y 45.0000, Z -5.5000, A 0.000, B 0.000, C 0.000 }
gfCNCPoint4[10027] = {X 60.1051, Y 44.2086, Z -5.5000, A 0.000, B 0.000, C 0.000 }
gfCNCPoint4[10028] = {X 60.1953, Y 43.3581, Z -5.5000, A 0.000, B 0.000, C 0.000 }
gfCNCPoint4[10029] = {X 60.4608, Y 42.5450, Z -5.5000, A 0.000, B 0.000, C 0.000 }
gfCNCPoint4[10030] = {X 60.8899, Y 41.8051, Z -5.5000, A 0.000, B 0.000, C 0.000 }
gfCNCPoint4[10031] = {X 60.1746, Y 39.8492, Z -5.5000, A 0.000, B 0.000, C 0.000 }
gfCNCPoint4[10032] = {X 51.9109, Y 39.8492, Z -5.5000, A 0.000, B 0.000, C 0.000 }
gfCNCPoint4[10033] = {X 51.0696, Y 42.1093, Z -5.5000, A 0.000, B 0.000, C 0.000 }
gfCNCPoint4[10034] = {X 51.1301, Y 42.2105, Z -5.5000, A 0.000, B 0.000, C 0.000 }
gfCNCPoint4[10035] = {X 51.4138, Y 42.8326, Z -5.5000, A 0.000, B 0.000, C 0.000 }
gfCNCPoint4[10036] = {X 51.5897, Y 43.4932, Z -5.5000, A 0.000, B 0.000, C 0.000 }
gfCNCPoint4[10037] = {X 51.6528, Y 44.1740, Z -5.5000, A 0.000, B 0.000, C 0.000 }
gfCNCPoint4[10038] = {X 51.6529, Y 45.0000, Z -5.5000, A 0.000, B 0.000, C 0.000 }
gfCNCPoint4[10039] = {X 51.5506, Y 45.9079, Z -5.5000, A 0.000, B 0.000, C 0.000 }
gfCNCPoint4[10040] = {X 51.2489, Y 46.7702, Z -5.5000, A 0.000, B 0.000, C 0.000 }
gfCNCPoint4[10041] = {X 50.7628, Y 47.5438, Z -5.5000, A 0.000, B 0.000, C 0.000 }
gfCNCPoint4[10042] = {X 50.1168, Y 48.1899, Z -5.5000, A 0.000, B 0.000, C 0.000 }
gfCNCPoint4[10043] = {X 49.3432, Y 48.6760, Z -5.5000, A 0.000, B 0.000, C 0.000 }
gfCNCPoint4[10044] = {X 48.4808, Y 48.9777, Z -5.5000, A 0.000, B 0.000, C 0.000 }
gfCNCPoint4[10045] = {X 47.5729, Y 49.0800, Z -5.5000, A 0.000, B 0.000, C 0.000 }
gfCNCPoint4[10046] = {X 40.6393, Y 49.0800, Z -5.5000, A 0.000, B 0.000, C 0.000 }
gfCNCPoint4[10047] = {X 39.7314, Y 48.9777, Z -5.5000, A 0.000, B 0.000, C 0.000 }
gfCNCPoint4[10048] = {X 38.8691, Y 48.6760, Z -5.5000, A 0.000, B 0.000, C 0.000 }
gfCNCPoint4[10049] = {X 38.0955, Y 48.1899, Z -5.5000, A 0.000, B 0.000, C 0.000 }
gfCNCPoint4[10050] = {X 37.4494, Y 47.5438, Z -5.5000, A 0.000, B 0.000, C 0.000 }
gfCNCPoint4[10051] = {X 36.9633, Y 46.7702, Z -5.5000, A 0.000, B 0.000, C 0.000 }
gfCNCPoint4[10052] = {X 36.6616, Y 45.9079, Z -5.5000, A 0.000, B 0.000, C 0.000 }
gfCNCPoint4[10053] = {X 36.5593, Y 45.0000, Z -5.5000, A 0.000, B 0.000, C 0.000 }
gfCNCPoint4[10054] = {X 36.5593, Y 44.2086, Z -5.5000, A 0.000, B 0.000, C 0.000 }
gfCNCPoint4[10055] = {X 36.6735, Y 43.2502, Z -5.5000, A 0.000, B 0.000, C 0.000 }
gfCNCPoint4[10056] = {X 37.0096, Y 42.3455, Z -5.5000, A 0.000, B 0.000, C 0.000 }
gfCNCPoint4[10057] = {X 37.5489, Y 41.5450, Z -5.5000, A 0.000, B 0.000, C 0.000 }
gfCNCPoint4[10058] = {X 38.2611, Y 40.8936, Z -5.5000, A 0.000, B 0.000, C 0.000 }
gfCNCPoint4[10059] = {X 39.1063, Y 40.4277, Z -5.5000, A 0.000, B 0.000, C 0.000 }
gfCNCPoint4[10060] = {X 39.1153, Y 40.4191, Z -5.5000, A 0.000, B 0.000, C 0.000 }
gfCNCPoint4[10061] = {X 39.1256, Y 40.3959, Z -5.5000, A 0.000, B 0.000, C 0.000 }
gfCNCPoint4[10062] = {X 39.7340, Y 38.9639, Z -5.5000, A 0.000, B 0.000, C 0.000 }
gfCNCPoint4[10063] = {X 40.2898, Y 37.5107, Z -5.5000, A 0.000, B 0.000, C 0.000 }
gfCNCPoint4[10064] = {X 43.8730, Y 27.8909, Z -5.5000, A 0.000, B 0.000, C 0.000 }
gfCNCPoint4[10065] = {X 40.1246, Y 26.4947, Z -5.5000, A 0.000, B 0.000, C 0.000 }
gfCNCPoint4[10066] = {X 43.9480, Y 27.9189, Z -5.5000, A 0.000, B 0.000, C 0.000 }
gfCNCPoint4[10067] = {X 48.6479, Y 15.3010, Z -5.5000, A 0.000, B 0.000, C 0.000 }
gfCNCPoint4[10068] = {X 48.2407, Y 14.5838, Z -5.5000, A 0.000, B 0.000, C 0.000 }
gfCNCPoint4[10069] = {X 47.9892, Y 13.7983, Z -5.5000, A 0.000, B 0.000, C 0.000 }
gfCNCPoint4[10070] = {X 47.9042, Y 12.9779, Z -5.5000, A 0.000, B 0.000, C 0.000 }
gfCNCPoint4[10071] = {X 47.9042, Y 12.1868, Z -5.5000, A 0.000, B 0.000, C 0.000 }
gfCNCPoint4[10072] = {X 48.0045, Y 11.2967, Z -5.5000, A 0.000, B 0.000, C 0.000 }
gfCNCPoint4[10073] = {X 48.3003, Y 10.4513, Z -5.5000, A 0.000, B 0.000, C 0.000 }
gfCNCPoint4[10074] = {X 48.7769, Y 9.6929, Z -5.5000, A 0.000, B 0.000, C 0.000 }
gfCNCPoint4[10075] = {X 49.4103, Y 9.0595, Z -5.5000, A 0.000, B 0.000, C 0.000 }
gfCNCPoint4[10076] = {X 50.1687, Y 8.5829, Z -5.5000, A 0.000, B 0.000, C 0.000 }
gfCNCPoint4[10077] = {X 51.0141, Y 8.2871, Z -5.5000, A 0.000, B 0.000, C 0.000 }
gfCNCPoint4[10078] = {X 51.9042, Y 8.1868, Z -5.5000, A 0.000, B 0.000, C 0.000 }
gfCNCPoint4[10079] = {X 59.6221, Y 8.1868, Z -5.5000, A 0.000, B 0.000, C 0.000 }
gfCNCPoint4[10080] = {X 60.5122, Y 8.2871, Z -5.5000, A 0.000, B 0.000, C 0.000 }
gfCNCPoint4[10081] = {X 61.3577, Y 8.5829, Z -5.5000, A 0.000, B 0.000, C 0.000 }
gfCNCPoint4[10082] = {X 62.1161, Y 9.0595, Z -5.5000, A 0.000, B 0.000, C 0.000 }
gfCNCPoint4[10083] = {X 62.7495, Y 9.6929, Z -5.5000, A 0.000, B 0.000, C 0.000 }
gfCNCPoint4[10084] = {X 63.2260, Y 10.4513, Z -5.5000, A 0.000, B 0.000, C 0.000 }
gfCNCPoint4[10085] = {X 63.5218, Y 11.2967, Z -5.5000, A 0.000, B 0.000, C 0.000 }
gfCNCPoint4[10086] = {X 63.6221, Y 12.1868, Z -5.5000, A 0.000, B 0.000, C 0.000 }
gfCNCPoint4[10087] = {X 63.6219, Y 13.0192, Z -5.5000, A 0.000, B 0.000, C 0.000 }
gfCNCPoint4[10088] = {X 63.5277, Y 13.8418, Z -5.5000, A 0.000, B 0.000, C 0.000 }
gfCNCPoint4[10089] = {X 63.2662, Y 14.6274, Z -5.5000, A 0.000, B 0.000, C 0.000 }
gfCNCPoint4[10090] = {X 62.8486, Y 15.3423, Z -5.5000, A 0.000, B 0.000, C 0.000 }
gfCNCPoint4[10091] = {X 63.1268, Y 16.0764, Z -5.5000, A 0.000, B 0.000, C 0.000 }
gfCNCPoint4[10092] = {X 65.9404, Y 23.5429, Z -5.5000, A 0.000, B 0.000, C 0.000 }
gfCNCPoint4[10093] = {X 71.9113, Y 39.6152, Z -5.5000, A 0.000, B 0.000, C 0.000 }
gfCNCPoint4[10094] = {X 72.2614, Y 40.4958, Z -5.5000, A 0.000, B 0.000, C 0.000 }
gfCNCPoint4[10095] = {X 72.2809, Y 40.5156, Z -5.5000, A 0.000, B 0.000, C 0.000 }
gfCNCPoint4[10096] = {X 72.3463, Y 40.5435, Z -5.5000, A 0.000, B 0.000, C 0.000 }
gfCNCPoint4[10097] = {X 72.4111, Y 40.5726, Z -5.5000, A 0.000, B 0.000, C 0.000 }
gfCNCPoint4[10098] = {X 73.1906, Y 41.0439, Z -5.5000, A 0.000, B 0.000, C 0.000 }
gfCNCPoint4[10099] = {X 73.8431, Y 41.6793, Z -5.5000, A 0.000, B 0.000, C 0.000 }
gfCNCPoint4[10100] = {X 74.3351, Y 42.4459, Z -5.5000, A 0.000, B 0.000, C 0.000 }
gfCNCPoint4[10101] = {X 74.6408, Y 43.3040, Z -5.5000, A 0.000, B 0.000, C 0.000 }
gfCNCPoint4[10102] = {X 74.7445, Y 44.2089, Z -5.5000, A 0.000, B 0.000, C 0.000 }
gfCNCPoint4[10103] = {X 74.7445, Y 45.0000, Z -5.5000, A 0.000, B 0.000, C 0.000 }
gfCNCPoint4[10104] = {X 74.6442, Y 45.8901, Z -5.5000, A 0.000, B 0.000, C 0.000 }
gfCNCPoint4[10105] = {X 74.3483, Y 46.7355, Z -5.5000, A 0.000, B 0.000, C 0.000 }
gfCNCPoint4[10106] = {X 73.8718, Y 47.4940, Z -5.5000, A 0.000, B 0.000, C 0.000 }
gfCNCPoint4[10107] = {X 73.2384, Y 48.1273, Z -5.5000, A 0.000, B 0.000, C 0.000 }
gfCNCPoint4[10108] = {X 72.4800, Y 48.6039, Z -5.5000, A 0.000, B 0.000, C 0.000 }
gfCNCPoint4[10109] = {X 71.6345, Y 48.8997, Z -5.5000, A 0.000, B 0.000, C 0.000 }
gfCNCPoint4[10110] = {X 70.7445, Y 49.0000, Z -5.5000, A 0.000, B 0.000, C 0.000 }
gfCNCPoint4[10111] = {X 64.1851, Y 49.0000, Z -5.5000, A 0.000, B 0.000, C 0.000 }
gfCNCPoint4[10112] = {X 63.2951, Y 48.8997, Z -5.5000, A 0.000, B 0.000, C 0.000 }
gfCNCPoint4[10113] = {X 62.4496, Y 48.6039, Z -5.5000, A 0.000, B 0.000, C 0.000 }
gfCNCPoint4[10114] = {X 61.6912, Y 48.1273, Z -5.5000, A 0.000, B 0.000, C 0.000 }
gfCNCPoint4[10115] = {X 61.0578, Y 47.4940, Z -5.5000, A 0.000, B 0.000, C 0.000 }
gfCNCPoint4[10116] = {X 60.5813, Y 46.7355, Z -5.5000, A 0.000, B 0.000, C 0.000 }
gfCNCPoint4[10117] = {X 60.2854, Y 45.8901, Z -5.5000, A 0.000, B 0.000, C 0.000 }
gfCNCPoint4[10118] = {X 60.1851, Y 45.0000, Z -5.5000, A 0.000, B 0.000, C 0.000 }
gfCNCPoint4[10119] = {X 60.1855, Y 44.1538, Z -5.5000, A 0.000, B 0.000, C 0.000 }
gfCNCPoint4[10120] = {X 60.2746, Y 43.3674, Z -5.5000, A 0.000, B 0.000, C 0.000 }
gfCNCPoint4[10121] = {X 60.5168, Y 42.6140, Z -5.5000, A 0.000, B 0.000, C 0.000 }
gfCNCPoint4[10122] = {X 60.9025, Y 41.9231, Z -5.5000, A 0.000, B 0.000, C 0.000 }
gfCNCPoint4[10123] = {X 60.9798, Y 41.8180, Z -5.5000, A 0.000, B 0.000, C 0.000 }
gfCNCPoint4[10124] = {X 60.2305, Y 39.7692, Z -5.5000, A 0.000, B 0.000, C 0.000 }
gfCNCPoint4[10125] = {X 51.8426, Y 39.7692, Z -5.5000, A 0.000, B 0.000, C 0.000 }
gfCNCPoint4[10126] = {X 51.8426, Y 39.8032, Z -5.5000, A 0.000, B 0.000, C 0.000 }
gfCNCPoint4[10127] = {X 50.9813, Y 42.1174, Z -5.5000, A 0.000, B 0.000, C 0.000 }
gfCNCPoint4[10128] = {X 51.0727, Y 42.2719, Z -5.5000, A 0.000, B 0.000, C 0.000 }
gfCNCPoint4[10129] = {X 51.3480, Y 42.8862, Z -5.5000, A 0.000, B 0.000, C 0.000 }
gfCNCPoint4[10130] = {X 51.5163, Y 43.5381, Z -5.5000, A 0.000, B 0.000, C 0.000 }
gfCNCPoint4[10131] = {X 51.5729, Y 44.2089, Z -5.5000, A 0.000, B 0.000, C 0.000 }
gfCNCPoint4[10132] = {X 51.5729, Y 45.0000, Z -5.5000, A 0.000, B 0.000, C 0.000 }
gfCNCPoint4[10133] = {X 51.4726, Y 45.8901, Z -5.5000, A 0.000, B 0.000, C 0.000 }
gfCNCPoint4[10134] = {X 51.1768, Y 46.7355, Z -5.5000, A 0.000, B 0.000, C 0.000 }
gfCNCPoint4[10135] = {X 50.7003, Y 47.4940, Z -5.5000, A 0.000, B 0.000, C 0.000 }
gfCNCPoint4[10136] = {X 50.0669, Y 48.1273, Z -5.5000, A 0.000, B 0.000, C 0.000 }
gfCNCPoint4[10137] = {X 49.3085, Y 48.6039, Z -5.5000, A 0.000, B 0.000, C 0.000 }
gfCNCPoint4[10138] = {X 48.4630, Y 48.8997, Z -5.5000, A 0.000, B 0.000, C 0.000 }
gfCNCPoint4[10139] = {X 47.5729, Y 49.0000, Z -5.5000, A 0.000, B 0.000, C 0.000 }
gfCNCPoint4[10140] = {X 40.6393, Y 49.0000, Z -5.5000, A 0.000, B 0.000, C 0.000 }
gfCNCPoint4[10141] = {X 39.7492, Y 48.8997, Z -5.5000, A 0.000, B 0.000, C 0.000 }
gfCNCPoint4[10142] = {X 38.9038, Y 48.6039, Z -5.5000, A 0.000, B 0.000, C 0.000 }
gfCNCPoint4[10143] = {X 38.1453, Y 48.1273, Z -5.5000, A 0.000, B 0.000, C 0.000 }
gfCNCPoint4[10144] = {X 37.5120, Y 47.4940, Z -5.5000, A 0.000, B 0.000, C 0.000 }
gfCNCPoint4[10145] = {X 37.0354, Y 46.7355, Z -5.5000, A 0.000, B 0.000, C 0.000 }
gfCNCPoint4[10146] = {X 36.7396, Y 45.8901, Z -5.5000, A 0.000, B 0.000, C 0.000 }
gfCNCPoint4[10147] = {X 36.6393, Y 45.0000, Z -5.5000, A 0.000, B 0.000, C 0.000 }
gfCNCPoint4[10148] = {X 36.6397, Y 44.1538, Z -5.5000, A 0.000, B 0.000, C 0.000 }
gfCNCPoint4[10149] = {X 36.7563, Y 43.2483, Z -5.5000, A 0.000, B 0.000, C 0.000 }
gfCNCPoint4[10150] = {X 37.0752, Y 42.3929, Z -5.5000, A 0.000, B 0.000, C 0.000 }
gfCNCPoint4[10151] = {X 37.5798, Y 41.6321, Z -5.5000, A 0.000, B 0.000, C 0.000 }
gfCNCPoint4[10152] = {X 38.2437, Y 41.0055, Z -5.5000, A 0.000, B 0.000, C 0.000 }
gfCNCPoint4[10153] = {X 39.0324, Y 40.5457, Z -5.5000, A 0.000, B 0.000, C 0.000 }
gfCNCPoint4[10154] = {X 39.0842, Y 40.5234, Z -5.5000, A 0.000, B 0.000, C 0.000 }
gfCNCPoint4[10155] = {X 39.1364, Y 40.5019, Z -5.5000, A 0.000, B 0.000, C 0.000 }
gfCNCPoint4[10156] = {X 39.1672, Y 40.4818, Z -5.5000, A 0.000, B 0.000, C 0.000 }
gfCNCPoint4[10157] = {X 39.1883, Y 40.4518, Z -5.5000, A 0.000, B 0.000, C 0.000 }
gfCNCPoint4[10158] = {X 39.2128, Y 40.3968, Z -5.5000, A 0.000, B 0.000, C 0.000 }
gfCNCPoint4[10159] = {X 39.2373, Y 40.3417, Z -5.5000, A 0.000, B 0.000, C 0.000 }
gfCNCPoint4[10160] = {X 39.8259, Y 38.9500, Z -5.5000, A 0.000, B 0.000, C 0.000 }
gfCNCPoint4[10161] = {X 40.3649, Y 37.5383, Z -5.5000, A 0.000, B 0.000, C 0.000 }
gfCNCPoint4[10162] = {X 43.9480, Y 27.9189, Z -5.5000, A 0.000, B 0.000, C 0.000 }
gfCNCPoint4[10163] = {X 40.1246, Y 26.4947, Z -5.5000, A 0.000, B 0.000, C 0.000 }
gfCNCPoint4[10164] = {X 40.1246, Y 26.4947, Z -2.5000, A 0.000, B 0.000, C 0.000 }
gfCNCPoint4[10165] = {X 40.1246, Y 26.4947, Z 11.0000, A 0.000, B 0.000, C 0.000 }
gfCNCPoint4[10166] = {X 79.0223, Y 28.5914, Z 11.0000, A 0.000, B 0.000, C 0.000 }
gfCNCPoint4[10167] = {X 79.0223, Y 28.5914, Z -2.5000, A 0.000, B 0.000, C 0.000 }
gfCNCPoint4[10168] = {X 79.0223, Y 28.5914, Z -5.5000, A 0.000, B 0.000, C 0.000 }
gfCNCPoint4[10169] = {X 83.1023, Y 28.5914, Z -5.5000, A 0.000, B 0.000, C 0.000 }
gfCNCPoint4[10170] = {X 83.1022, Y 16.2738, Z -5.5000, A 0.000, B 0.000, C 0.000 }
gfCNCPoint4[10171] = {X 82.4638, Y 15.6027, Z -5.5000, A 0.000, B 0.000, C 0.000 }
gfCNCPoint4[10172] = {X 81.9832, Y 14.8110, Z -5.5000, A 0.000, B 0.000, C 0.000 }
gfCNCPoint4[10173] = {X 81.6824, Y 13.9350, Z -5.5000, A 0.000, B 0.000, C 0.000 }
gfCNCPoint4[10174] = {X 81.5752, Y 13.0150, Z -5.5000, A 0.000, B 0.000, C 0.000 }
gfCNCPoint4[10175] = {X 81.5751, Y 12.1868, Z -5.5000, A 0.000, B 0.000, C 0.000 }
gfCNCPoint4[10176] = {X 81.6834, Y 11.2255, Z -5.5000, A 0.000, B 0.000, C 0.000 }
gfCNCPoint4[10177] = {X 82.0029, Y 10.3125, Z -5.5000, A 0.000, B 0.000, C 0.000 }
gfCNCPoint4[10178] = {X 82.5176, Y 9.4933, Z -5.5000, A 0.000, B 0.000, C 0.000 }
gfCNCPoint4[10179] = {X 83.2016, Y 8.8093, Z -5.5000, A 0.000, B 0.000, C 0.000 }
gfCNCPoint4[10180] = {X 84.0207, Y 8.2946, Z -5.5000, A 0.000, B 0.000, C 0.000 }
gfCNCPoint4[10181] = {X 84.9338, Y 7.9751, Z -5.5000, A 0.000, B 0.000, C 0.000 }
gfCNCPoint4[10182] = {X 85.8951, Y 7.8668, Z -5.5000, A 0.000, B 0.000, C 0.000 }
gfCNCPoint4[10183] = {X 94.0497, Y 7.8668, Z -5.5000, A 0.000, B 0.000, C 0.000 }
gfCNCPoint4[10184] = {X 95.0110, Y 7.9751, Z -5.5000, A 0.000, B 0.000, C 0.000 }
gfCNCPoint4[10185] = {X 95.9240, Y 8.2946, Z -5.5000, A 0.000, B 0.000, C 0.000 }
gfCNCPoint4[10186] = {X 96.7431, Y 8.8093, Z -5.5000, A 0.000, B 0.000, C 0.000 }
gfCNCPoint4[10187] = {X 97.4272, Y 9.4933, Z -5.5000, A 0.000, B 0.000, C 0.000 }
gfCNCPoint4[10188] = {X 97.9419, Y 10.3124, Z -5.5000, A 0.000, B 0.000, C 0.000 }
gfCNCPoint4[10189] = {X 98.2614, Y 11.2255, Z -5.5000, A 0.000, B 0.000, C 0.000 }
gfCNCPoint4[10190] = {X 98.3697, Y 12.1868, Z -5.5000, A 0.000, B 0.000, C 0.000 }
gfCNCPoint4[10191] = {X 98.3697, Y 12.9782, Z -5.5000, A 0.000, B 0.000, C 0.000 }
gfCNCPoint4[10192] = {X 98.2967, Y 13.7679, Z -5.5000, A 0.000, B 0.000, C 0.000 }
gfCNCPoint4[10193] = {X 98.0806, Y 14.5310, Z -5.5000, A 0.000, B 0.000, C 0.000 }
gfCNCPoint4[10194] = {X 97.7287, Y 15.2417, Z -5.5000, A 0.000, B 0.000, C 0.000 }
gfCNCPoint4[10195] = {X 101.8759, Y 25.5234, Z -5.5000, A 0.000, B 0.000, C 0.000 }
gfCNCPoint4[10196] = {X 106.0163, Y 15.2212, Z -5.5000, A 0.000, B 0.000, C 0.000 }
gfCNCPoint4[10197] = {X 105.6761, Y 14.5284, Z -5.5000, A 0.000, B 0.000, C 0.000 }
gfCNCPoint4[10198] = {X 105.4645, Y 13.7860, Z -5.5000, A 0.000, B 0.000, C 0.000 }
gfCNCPoint4[10199] = {X 105.3885, Y 13.0179, Z -5.5000, A 0.000, B 0.000, C 0.000 }
gfCNCPoint4[10200] = {X 105.3883, Y 12.1868, Z -5.5000, A 0.000, B 0.000, C 0.000 }
gfCNCPoint4[10201] = {X 105.4966, Y 11.2255, Z -5.5000, A 0.000, B 0.000, C 0.000 }
gfCNCPoint4[10202] = {X 105.8161, Y 10.3124, Z -5.5000, A 0.000, B 0.000, C 0.000 }
gfCNCPoint4[10203] = {X 106.3308, Y 9.4933, Z -5.5000, A 0.000, B 0.000, C 0.000 }
gfCNCPoint4[10204] = {X 107.0148, Y 8.8093, Z -5.5000, A 0.000, B 0.000, C 0.000 }
gfCNCPoint4[10205] = {X 107.8339, Y 8.2946, Z -5.5000, A 0.000, B 0.000, C 0.000 }
gfCNCPoint4[10206] = {X 108.7470, Y 7.9751, Z -5.5000, A 0.000, B 0.000, C 0.000 }
gfCNCPoint4[10207] = {X 109.7083, Y 7.8668, Z -5.5000, A 0.000, B 0.000, C 0.000 }
gfCNCPoint4[10208] = {X 117.7916, Y 7.8668, Z -5.5000, A 0.000, B 0.000, C 0.000 }
gfCNCPoint4[10209] = {X 118.7529, Y 7.9751, Z -5.5000, A 0.000, B 0.000, C 0.000 }
gfCNCPoint4[10210] = {X 119.6660, Y 8.2946, Z -5.5000, A 0.000, B 0.000, C 0.000 }
gfCNCPoint4[10211] = {X 120.4851, Y 8.8093, Z -5.5000, A 0.000, B 0.000, C 0.000 }
gfCNCPoint4[10212] = {X 121.1691, Y 9.4933, Z -5.5000, A 0.000, B 0.000, C 0.000 }
gfCNCPoint4[10213] = {X 121.6838, Y 10.3124, Z -5.5000, A 0.000, B 0.000, C 0.000 }
gfCNCPoint4[10214] = {X 122.0033, Y 11.2255, Z -5.5000, A 0.000, B 0.000, C 0.000 }
gfCNCPoint4[10215] = {X 122.1116, Y 12.1868, Z -5.5000, A 0.000, B 0.000, C 0.000 }
gfCNCPoint4[10216] = {X 122.1116, Y 12.9782, Z -5.5000, A 0.000, B 0.000, C 0.000 }
gfCNCPoint4[10217] = {X 122.0103, Y 13.9078, Z -5.5000, A 0.000, B 0.000, C 0.000 }
gfCNCPoint4[10218] = {X 121.7114, Y 14.7939, Z -5.5000, A 0.000, B 0.000, C 0.000 }
gfCNCPoint4[10219] = {X 121.2288, Y 15.5949, Z -5.5000, A 0.000, B 0.000, C 0.000 }
gfCNCPoint4[10220] = {X 120.5851, Y 16.2732, Z -5.5000, A 0.000, B 0.000, C 0.000 }
gfCNCPoint4[10221] = {X 120.5844, Y 40.9143, Z -5.5000, A 0.000, B 0.000, C 0.000 }
gfCNCPoint4[10222] = {X 120.6224, Y 40.9456, Z -5.5000, A 0.000, B 0.000, C 0.000 }
gfCNCPoint4[10223] = {X 121.2457, Y 41.6143, Z -5.5000, A 0.000, B 0.000, C 0.000 }
gfCNCPoint4[10224] = {X 121.7143, Y 42.3992, Z -5.5000, A 0.000, B 0.000, C 0.000 }
gfCNCPoint4[10225] = {X 122.0073, Y 43.2652, Z -5.5000, A 0.000, B 0.000, C 0.000 }
gfCNCPoint4[10226] = {X 122.1114, Y 44.1734, Z -5.5000, A 0.000, B 0.000, C 0.000 }
gfCNCPoint4[10227] = {X 122.1116, Y 45.0000, Z -5.5000, A 0.000, B 0.000, C 0.000 }
gfCNCPoint4[10228] = {X 122.0033, Y 45.9613, Z -5.5000, A 0.000, B 0.000, C 0.000 }
gfCNCPoint4[10229] = {X 121.6838, Y 46.8744, Z -5.5000, A 0.000, B 0.000, C 0.000 }
gfCNCPoint4[10230] = {X 121.1691, Y 47.6935, Z -5.5000, A 0.000, B 0.000, C 0.000 }
gfCNCPoint4[10231] = {X 120.4851, Y 48.3775, Z -5.5000, A 0.000, B 0.000, C 0.000 }
gfCNCPoint4[10232] = {X 119.6660, Y 48.8922, Z -5.5000, A 0.000, B 0.000, C 0.000 }
gfCNCPoint4[10233] = {X 118.7529, Y 49.2117, Z -5.5000, A 0.000, B 0.000, C 0.000 }
gfCNCPoint4[10234] = {X 117.7916, Y 49.3200, Z -5.5000, A 0.000, B 0.000, C 0.000 }
gfCNCPoint4[10235] = {X 111.9185, Y 49.3200, Z -5.5000, A 0.000, B 0.000, C 0.000 }
gfCNCPoint4[10236] = {X 110.9619, Y 49.2128, Z -5.5000, A 0.000, B 0.000, C 0.000 }
gfCNCPoint4[10237] = {X 110.0529, Y 48.8964, Z -5.5000, A 0.000, B 0.000, C 0.000 }
gfCNCPoint4[10238] = {X 109.2365, Y 48.3866, Z -5.5000, A 0.000, B 0.000, C 0.000 }
gfCNCPoint4[10239] = {X 108.5532, Y 47.7087, Z -5.5000, A 0.000, B 0.000, C 0.000 }
gfCNCPoint4[10240] = {X 108.0369, Y 46.8963, Z -5.5000, A 0.000, B 0.000, C 0.000 }
gfCNCPoint4[10241] = {X 107.7134, Y 45.9898, Z -5.5000, A 0.000, B 0.000, C 0.000 }
gfCNCPoint4[10242] = {X 107.5986, Y 45.0341, Z -5.5000, A 0.000, B 0.000, C 0.000 }
gfCNCPoint4[10243] = {X 107.5985, Y 44.1807, Z -5.5000, A 0.000, B 0.000, C 0.000 }
gfCNCPoint4[10244] = {X 107.6343, Y 43.6363, Z -5.5000, A 0.000, B 0.000, C 0.000 }
gfCNCPoint4[10245] = {X 107.7409, Y 43.1012, Z -5.5000, A 0.000, B 0.000, C 0.000 }
gfCNCPoint4[10246] = {X 107.9085, Y 42.6047, Z -5.5000, A 0.000, B 0.000, C 0.000 }
gfCNCPoint4[10247] = {X 108.1371, Y 42.1332, Z -5.5000, A 0.000, B 0.000, C 0.000 }
gfCNCPoint4[10248] = {X 108.5871, Y 41.4634, Z -5.5000, A 0.000, B 0.000, C 0.000 }
gfCNCPoint4[10249] = {X 109.1256, Y 40.8623, Z -5.5000, A 0.000, B 0.000, C 0.000 }
gfCNCPoint4[10250] = {X 109.1255, Y 39.2969, Z -5.5000, A 0.000, B 0.000, C 0.000 }
gfCNCPoint4[10251] = {X 106.1118, Y 46.6615, Z -5.5000, A 0.000, B 0.000, C 0.000 }
gfCNCPoint4[10252] = {X 105.7417, Y 47.3611, Z -5.5000, A 0.000, B 0.000, C 0.000 }
gfCNCPoint4[10253] = {X 105.2502, Y 47.9815, Z -5.5000, A 0.000, B 0.000, C 0.000 }
gfCNCPoint4[10254] = {X 104.6538, Y 48.5018, Z -5.5000, A 0.000, B 0.000, C 0.000 }
gfCNCPoint4[10255] = {X 103.9724, Y 48.9046, Z -5.5000, A 0.000, B 0.000, C 0.000 }
gfCNCPoint4[10256] = {X 103.0287, Y 49.2242, Z -5.5000, A 0.000, B 0.000, C 0.000 }
gfCNCPoint4[10257] = {X 102.0368, Y 49.3191, Z -5.5000, A 0.000, B 0.000, C 0.000 }
gfCNCPoint4[10258] = {X 101.0496, Y 49.1842, Z -5.5000, A 0.000, B 0.000, C 0.000 }
gfCNCPoint4[10259] = {X 100.1195, Y 48.8268, Z -5.5000, A 0.000, B 0.000, C 0.000 }
gfCNCPoint4[10260] = {X 99.2961, Y 48.2657, Z -5.5000, A 0.000, B 0.000, C 0.000 }
gfCNCPoint4[10261] = {X 98.6231, Y 47.5309, Z -5.5000, A 0.000, B 0.000, C 0.000 }
gfCNCPoint4[10262] = {X 98.1363, Y 46.6615, Z -5.5000, A 0.000, B 0.000, C 0.000 }
gfCNCPoint4[10263] = {X 95.1314, Y 39.3125, Z -5.5000, A 0.000, B 0.000, C 0.000 }
gfCNCPoint4[10264] = {X 95.1314, Y 40.9049, Z -5.5000, A 0.000, B 0.000, C 0.000 }
gfCNCPoint4[10265] = {X 95.6580, Y 41.4443, Z -5.5000, A 0.000, B 0.000, C 0.000 }
gfCNCPoint4[10266] = {X 96.0849, Y 42.0655, Z -5.5000, A 0.000, B 0.000, C 0.000 }
gfCNCPoint4[10267] = {X 96.3312, Y 42.5726, Z -5.5000, A 0.000, B 0.000, C 0.000 }
gfCNCPoint4[10268] = {X 96.5107, Y 43.1069, Z -5.5000, A 0.000, B 0.000, C 0.000 }
gfCNCPoint4[10269] = {X 96.6194, Y 43.6521, Z -5.5000, A 0.000, B 0.000, C 0.000 }
gfCNCPoint4[10270] = {X 96.6585, Y 44.2065, Z -5.5000, A 0.000, B 0.000, C 0.000 }
gfCNCPoint4[10271] = {X 96.6583, Y 45.0415, Z -5.5000, A 0.000, B 0.000, C 0.000 }
gfCNCPoint4[10272] = {X 96.5422, Y 45.9960, Z -5.5000, A 0.000, B 0.000, C 0.000 }
gfCNCPoint4[10273] = {X 96.2178, Y 46.9011, Z -5.5000, A 0.000, B 0.000, C 0.000 }
gfCNCPoint4[10274] = {X 95.7012, Y 47.7120, Z -5.5000, A 0.000, B 0.000, C 0.000 }
gfCNCPoint4[10275] = {X 95.0181, Y 48.3886, Z -5.5000, A 0.000, B 0.000, C 0.000 }
gfCNCPoint4[10276] = {X 94.2022, Y 48.8973, Z -5.5000, A 0.000, B 0.000, C 0.000 }
gfCNCPoint4[10277] = {X 93.2940, Y 49.2130, Z -5.5000, A 0.000, B 0.000, C 0.000 }
gfCNCPoint4[10278] = {X 92.3385, Y 49.3200, Z -5.5000, A 0.000, B 0.000, C 0.000 }
gfCNCPoint4[10279] = {X 85.8951, Y 49.3200, Z -5.5000, A 0.000, B 0.000, C 0.000 }
gfCNCPoint4[10280] = {X 84.9387, Y 49.2128, Z -5.5000, A 0.000, B 0.000, C 0.000 }
gfCNCPoint4[10281] = {X 84.0297, Y 48.8965, Z -5.5000, A 0.000, B 0.000, C 0.000 }
gfCNCPoint4[10282] = {X 83.2134, Y 48.3869, Z -5.5000, A 0.000, B 0.000, C 0.000 }
gfCNCPoint4[10283] = {X 82.5301, Y 47.7091, Z -5.5000, A 0.000, B 0.000, C 0.000 }
gfCNCPoint4[10284] = {X 82.0138, Y 46.8970, Z -5.5000, A 0.000, B 0.000, C 0.000 }
gfCNCPoint4[10285] = {X 81.6902, Y 45.9906, Z -5.5000, A 0.000, B 0.000, C 0.000 }
gfCNCPoint4[10286] = {X 81.5752, Y 45.0351, Z -5.5000, A 0.000, B 0.000, C 0.000 }
gfCNCPoint4[10287] = {X 81.5751, Y 44.2071, Z -5.5000, A 0.000, B 0.000, C 0.000 }
gfCNCPoint4[10288] = {X 81.6801, Y 43.2778, Z -5.5000, A 0.000, B 0.000, C 0.000 }
gfCNCPoint4[10289] = {X 81.9802, Y 42.3920, Z -5.5000, A 0.000, B 0.000, C 0.000 }
gfCNCPoint4[10290] = {X 82.4617, Y 41.5901, Z -5.5000, A 0.000, B 0.000, C 0.000 }
gfCNCPoint4[10291] = {X 83.1025, Y 40.9089, Z -5.5000, A 0.000, B 0.000, C 0.000 }
gfCNCPoint4[10292] = {X 83.1023, Y 28.5914, Z -5.5000, A 0.000, B 0.000, C 0.000 }
gfCNCPoint4[10293] = {X 79.1023, Y 28.5914, Z -5.5000, A 0.000, B 0.000, C 0.000 }
gfCNCPoint4[10294] = {X 83.1823, Y 28.5914, Z -5.5000, A 0.000, B 0.000, C 0.000 }
gfCNCPoint4[10295] = {X 83.1822, Y 16.2365, Z -5.5000, A 0.000, B 0.000, C 0.000 }
gfCNCPoint4[10296] = {X 82.5443, Y 15.5761, Z -5.5000, A 0.000, B 0.000, C 0.000 }
gfCNCPoint4[10297] = {X 82.0635, Y 14.7937, Z -5.5000, A 0.000, B 0.000, C 0.000 }
gfCNCPoint4[10298] = {X 81.7625, Y 13.9262, Z -5.5000, A 0.000, B 0.000, C 0.000 }
gfCNCPoint4[10299] = {X 81.6552, Y 13.0143, Z -5.5000, A 0.000, B 0.000, C 0.000 }
gfCNCPoint4[10300] = {X 81.6551, Y 12.1868, Z -5.5000, A 0.000, B 0.000, C 0.000 }
gfCNCPoint4[10301] = {X 81.7614, Y 11.2433, Z -5.5000, A 0.000, B 0.000, C 0.000 }
gfCNCPoint4[10302] = {X 82.0750, Y 10.3472, Z -5.5000, A 0.000, B 0.000, C 0.000 }
gfCNCPoint4[10303] = {X 82.5801, Y 9.5432, Z -5.5000, A 0.000, B 0.000, C 0.000 }
gfCNCPoint4[10304] = {X 83.2515, Y 8.8719, Z -5.5000, A 0.000, B 0.000, C 0.000 }
gfCNCPoint4[10305] = {X 84.0554, Y 8.3667, Z -5.5000, A 0.000, B 0.000, C 0.000 }
gfCNCPoint4[10306] = {X 84.9516, Y 8.0531, Z -5.5000, A 0.000, B 0.000, C 0.000 }
gfCNCPoint4[10307] = {X 85.8951, Y 7.9468, Z -5.5000, A 0.000, B 0.000, C 0.000 }
gfCNCPoint4[10308] = {X 94.0497, Y 7.9468, Z -5.5000, A 0.000, B 0.000, C 0.000 }
gfCNCPoint4[10309] = {X 94.9932, Y 8.0531, Z -5.5000, A 0.000, B 0.000, C 0.000 }
gfCNCPoint4[10310] = {X 95.8893, Y 8.3667, Z -5.5000, A 0.000, B 0.000, C 0.000 }
gfCNCPoint4[10311] = {X 96.6933, Y 8.8718, Z -5.5000, A 0.000, B 0.000, C 0.000 }
gfCNCPoint4[10312] = {X 97.3646, Y 9.5432, Z -5.5000, A 0.000, B 0.000, C 0.000 }
gfCNCPoint4[10313] = {X 97.8698, Y 10.3471, Z -5.5000, A 0.000, B 0.000, C 0.000 }
gfCNCPoint4[10314] = {X 98.1834, Y 11.2433, Z -5.5000, A 0.000, B 0.000, C 0.000 }
gfCNCPoint4[10315] = {X 98.2897, Y 12.1868, Z -5.5000, A 0.000, B 0.000, C 0.000 }
gfCNCPoint4[10316] = {X 98.2897, Y 12.9782, Z -5.5000, A 0.000, B 0.000, C 0.000 }
gfCNCPoint4[10317] = {X 98.2156, Y 13.7664, Z -5.5000, A 0.000, B 0.000, C 0.000 }
gfCNCPoint4[10318] = {X 97.9962, Y 14.5272, Z -5.5000, A 0.000, B 0.000, C 0.000 }
gfCNCPoint4[10319] = {X 97.6393, Y 15.2339, Z -5.5000, A 0.000, B 0.000, C 0.000 }
gfCNCPoint4[10320] = {X 101.8760, Y 25.7375, Z -5.5000, A 0.000, B 0.000, C 0.000 }
gfCNCPoint4[10321] = {X 106.1056, Y 15.2137, Z -5.5000, A 0.000, B 0.000, C 0.000 }
gfCNCPoint4[10322] = {X 105.7603, Y 14.5244, Z -5.5000, A 0.000, B 0.000, C 0.000 }
gfCNCPoint4[10323] = {X 105.5456, Y 13.7841, Z -5.5000, A 0.000, B 0.000, C 0.000 }
gfCNCPoint4[10324] = {X 105.4685, Y 13.0172, Z -5.5000, A 0.000, B 0.000, C 0.000 }
gfCNCPoint4[10325] = {X 105.4683, Y 12.1868, Z -5.5000, A 0.000, B 0.000, C 0.000 }
gfCNCPoint4[10326] = {X 105.5746, Y 11.2433, Z -5.5000, A 0.000, B 0.000, C 0.000 }
gfCNCPoint4[10327] = {X 105.8882, Y 10.3471, Z -5.5000, A 0.000, B 0.000, C 0.000 }
gfCNCPoint4[10328] = {X 106.3933, Y 9.5432, Z -5.5000, A 0.000, B 0.000, C 0.000 }
gfCNCPoint4[10329] = {X 107.0647, Y 8.8718, Z -5.5000, A 0.000, B 0.000, C 0.000 }
gfCNCPoint4[10330] = {X 107.8686, Y 8.3667, Z -5.5000, A 0.000, B 0.000, C 0.000 }
gfCNCPoint4[10331] = {X 108.7648, Y 8.0531, Z -5.5000, A 0.000, B 0.000, C 0.000 }
gfCNCPoint4[10332] = {X 109.7083, Y 7.9468, Z -5.5000, A 0.000, B 0.000, C 0.000 }
gfCNCPoint4[10333] = {X 117.7916, Y 7.9468, Z -5.5000, A 0.000, B 0.000, C 0.000 }
gfCNCPoint4[10334] = {X 118.7351, Y 8.0531, Z -5.5000, A 0.000, B 0.000, C 0.000 }
gfCNCPoint4[10335] = {X 119.6312, Y 8.3667, Z -5.5000, A 0.000, B 0.000, C 0.000 }
gfCNCPoint4[10336] = {X 120.4352, Y 8.8718, Z -5.5000, A 0.000, B 0.000, C 0.000 }
gfCNCPoint4[10337] = {X 121.1065, Y 9.5432, Z -5.5000, A 0.000, B 0.000, C 0.000 }
gfCNCPoint4[10338] = {X 121.6117, Y 10.3471, Z -5.5000, A 0.000, B 0.000, C 0.000 }
gfCNCPoint4[10339] = {X 121.9253, Y 11.2433, Z -5.5000, A 0.000, B 0.000, C 0.000 }
gfCNCPoint4[10340] = {X 122.0316, Y 12.1868, Z -5.5000, A 0.000, B 0.000, C 0.000 }
gfCNCPoint4[10341] = {X 122.0316, Y 12.9782, Z -5.5000, A 0.000, B 0.000, C 0.000 }
gfCNCPoint4[10342] = {X 121.9302, Y 13.8996, Z -5.5000, A 0.000, B 0.000, C 0.000 }
gfCNCPoint4[10343] = {X 121.6310, Y 14.7770, Z -5.5000, A 0.000, B 0.000, C 0.000 }
gfCNCPoint4[10344] = {X 121.1483, Y 15.5684, Z -5.5000, A 0.000, B 0.000, C 0.000 }
gfCNCPoint4[10345] = {X 120.5051, Y 16.2360, Z -5.5000, A 0.000, B 0.000, C 0.000 }
gfCNCPoint4[10346] = {X 120.5044, Y 40.9522, Z -5.5000, A 0.000, B 0.000, C 0.000 }
gfCNCPoint4[10347] = {X 120.5708, Y 41.0067, Z -5.5000, A 0.000, B 0.000, C 0.000 }
gfCNCPoint4[10348] = {X 121.1822, Y 41.6630, Z -5.5000, A 0.000, B 0.000, C 0.000 }
gfCNCPoint4[10349] = {X 121.6419, Y 42.4332, Z -5.5000, A 0.000, B 0.000, C 0.000 }
gfCNCPoint4[10350] = {X 121.9293, Y 43.2829, Z -5.5000, A 0.000, B 0.000, C 0.000 }
gfCNCPoint4[10351] = {X 122.0314, Y 44.1740, Z -5.5000, A 0.000, B 0.000, C 0.000 }
gfCNCPoint4[10352] = {X 122.0316, Y 45.0000, Z -5.5000, A 0.000, B 0.000, C 0.000 }
gfCNCPoint4[10353] = {X 121.9253, Y 45.9435, Z -5.5000, A 0.000, B 0.000, C 0.000 }
gfCNCPoint4[10354] = {X 121.6117, Y 46.8397, Z -5.5000, A 0.000, B 0.000, C 0.000 }
gfCNCPoint4[10355] = {X 121.1065, Y 47.6436, Z -5.5000, A 0.000, B 0.000, C 0.000 }
gfCNCPoint4[10356] = {X 120.4352, Y 48.3150, Z -5.5000, A 0.000, B 0.000, C 0.000 }
gfCNCPoint4[10357] = {X 119.6312, Y 48.8201, Z -5.5000, A 0.000, B 0.000, C 0.000 }
gfCNCPoint4[10358] = {X 118.7351, Y 49.1337, Z -5.5000, A 0.000, B 0.000, C 0.000 }
gfCNCPoint4[10359] = {X 117.7916, Y 49.2400, Z -5.5000, A 0.000, B 0.000, C 0.000 }
gfCNCPoint4[10360] = {X 111.9185, Y 49.2400, Z -5.5000, A 0.000, B 0.000, C 0.000 }
gfCNCPoint4[10361] = {X 110.9797, Y 49.1348, Z -5.5000, A 0.000, B 0.000, C 0.000 }
gfCNCPoint4[10362] = {X 110.0874, Y 48.8242, Z -5.5000, A 0.000, B 0.000, C 0.000 }
gfCNCPoint4[10363] = {X 109.2861, Y 48.3239, Z -5.5000, A 0.000, B 0.000, C 0.000 }
gfCNCPoint4[10364] = {X 108.6155, Y 47.6585, Z -5.5000, A 0.000, B 0.000, C 0.000 }
gfCNCPoint4[10365] = {X 108.1088, Y 46.8612, Z -5.5000, A 0.000, B 0.000, C 0.000 }
gfCNCPoint4[10366] = {X 107.7913, Y 45.9714, Z -5.5000, A 0.000, B 0.000, C 0.000 }
gfCNCPoint4[10367] = {X 107.6786, Y 45.0335, Z -5.5000, A 0.000, B 0.000, C 0.000 }
gfCNCPoint4[10368] = {X 107.6785, Y 44.1807, Z -5.5000, A 0.000, B 0.000, C 0.000 }
gfCNCPoint4[10369] = {X 107.7136, Y 43.6468, Z -5.5000, A 0.000, B 0.000, C 0.000 }
gfCNCPoint4[10370] = {X 107.8182, Y 43.1220, Z -5.5000, A 0.000, B 0.000, C 0.000 }
gfCNCPoint4[10371] = {X 107.9825, Y 42.6350, Z -5.5000, A 0.000, B 0.000, C 0.000 }
gfCNCPoint4[10372] = {X 108.2067, Y 42.1726, Z -5.5000, A 0.000, B 0.000, C 0.000 }
gfCNCPoint4[10373] = {X 108.6608, Y 41.4990, Z -5.5000, A 0.000, B 0.000, C 0.000 }
gfCNCPoint4[10374] = {X 109.2056, Y 40.8963, Z -5.5000, A 0.000, B 0.000, C 0.000 }
gfCNCPoint4[10375] = {X 109.2055, Y 39.1629, Z -5.5000, A 0.000, B 0.000, C 0.000 }
gfCNCPoint4[10376] = {X 109.0939, Y 39.1629, Z -5.5000, A 0.000, B 0.000, C 0.000 }
gfCNCPoint4[10377] = {X 106.0379, Y 46.6307, Z -5.5000, A 0.000, B 0.000, C 0.000 }
gfCNCPoint4[10378] = {X 105.6747, Y 47.3174, Z -5.5000, A 0.000, B 0.000, C 0.000 }
gfCNCPoint4[10379] = {X 105.1923, Y 47.9263, Z -5.5000, A 0.000, B 0.000, C 0.000 }
gfCNCPoint4[10380] = {X 104.6069, Y 48.4370, Z -5.5000, A 0.000, B 0.000, C 0.000 }
gfCNCPoint4[10381] = {X 103.9382, Y 48.8323, Z -5.5000, A 0.000, B 0.000, C 0.000 }
gfCNCPoint4[10382] = {X 103.0119, Y 49.1460, Z -5.5000, A 0.000, B 0.000, C 0.000 }
gfCNCPoint4[10383] = {X 102.0384, Y 49.2391, Z -5.5000, A 0.000, B 0.000, C 0.000 }
gfCNCPoint4[10384] = {X 101.0695, Y 49.1068, Z -5.5000, A 0.000, B 0.000, C 0.000 }
gfCNCPoint4[10385] = {X 100.1566, Y 48.7559, Z -5.5000, A 0.000, B 0.000, C 0.000 }
gfCNCPoint4[10386] = {X 99.3484, Y 48.2052, Z -5.5000, A 0.000, B 0.000, C 0.000 }
gfCNCPoint4[10387] = {X 98.6879, Y 47.4840, Z -5.5000, A 0.000, B 0.000, C 0.000 }
gfCNCPoint4[10388] = {X 98.2102, Y 46.6307, Z -5.5000, A 0.000, B 0.000, C 0.000 }
gfCNCPoint4[10389] = {X 95.0513, Y 38.9054, Z -5.5000, A 0.000, B 0.000, C 0.000 }
gfCNCPoint4[10390] = {X 95.0514, Y 40.9418, Z -5.5000, A 0.000, B 0.000, C 0.000 }
gfCNCPoint4[10391] = {X 95.5846, Y 41.4810, Z -5.5000, A 0.000, B 0.000, C 0.000 }
gfCNCPoint4[10392] = {X 96.0153, Y 42.1050, Z -5.5000, A 0.000, B 0.000, C 0.000 }
gfCNCPoint4[10393] = {X 96.2571, Y 42.6028, Z -5.5000, A 0.000, B 0.000, C 0.000 }
gfCNCPoint4[10394] = {X 96.4334, Y 43.1275, Z -5.5000, A 0.000, B 0.000, C 0.000 }
gfCNCPoint4[10395] = {X 96.5401, Y 43.6627, Z -5.5000, A 0.000, B 0.000, C 0.000 }
gfCNCPoint4[10396] = {X 96.5785, Y 44.2071, Z -5.5000, A 0.000, B 0.000, C 0.000 }
gfCNCPoint4[10397] = {X 96.5783, Y 45.0408, Z -5.5000, A 0.000, B 0.000, C 0.000 }
gfCNCPoint4[10398] = {X 96.4643, Y 45.9775, Z -5.5000, A 0.000, B 0.000, C 0.000 }
gfCNCPoint4[10399] = {X 96.1459, Y 46.8659, Z -5.5000, A 0.000, B 0.000, C 0.000 }
gfCNCPoint4[10400] = {X 95.6389, Y 47.6618, Z -5.5000, A 0.000, B 0.000, C 0.000 }
gfCNCPoint4[10401] = {X 94.9685, Y 48.3258, Z -5.5000, A 0.000, B 0.000, C 0.000 }
gfCNCPoint4[10402] = {X 94.1677, Y 48.8251, Z -5.5000, A 0.000, B 0.000, C 0.000 }
gfCNCPoint4[10403] = {X 93.2764, Y 49.1350, Z -5.5000, A 0.000, B 0.000, C 0.000 }
gfCNCPoint4[10404] = {X 92.3385, Y 49.2400, Z -5.5000, A 0.000, B 0.000, C 0.000 }
gfCNCPoint4[10405] = {X 85.8951, Y 49.2400, Z -5.5000, A 0.000, B 0.000, C 0.000 }
gfCNCPoint4[10406] = {X 84.9564, Y 49.1348, Z -5.5000, A 0.000, B 0.000, C 0.000 }
gfCNCPoint4[10407] = {X 84.0643, Y 48.8244, Z -5.5000, A 0.000, B 0.000, C 0.000 }
gfCNCPoint4[10408] = {X 83.2631, Y 48.3242, Z -5.5000, A 0.000, B 0.000, C 0.000 }
gfCNCPoint4[10409] = {X 82.5924, Y 47.6590, Z -5.5000, A 0.000, B 0.000, C 0.000 }
gfCNCPoint4[10410] = {X 82.0857, Y 46.8618, Z -5.5000, A 0.000, B 0.000, C 0.000 }
gfCNCPoint4[10411] = {X 81.7681, Y 45.9723, Z -5.5000, A 0.000, B 0.000, C 0.000 }
gfCNCPoint4[10412] = {X 81.6552, Y 45.0345, Z -5.5000, A 0.000, B 0.000, C 0.000 }
gfCNCPoint4[10413] = {X 81.6551, Y 44.2075, Z -5.5000, A 0.000, B 0.000, C 0.000 }
gfCNCPoint4[10414] = {X 81.7602, Y 43.2862, Z -5.5000, A 0.000, B 0.000, C 0.000 }
gfCNCPoint4[10415] = {X 82.0606, Y 42.4090, Z -5.5000, A 0.000, B 0.000, C 0.000 }
gfCNCPoint4[10416] = {X 82.5421, Y 41.6165, Z -5.5000, A 0.000, B 0.000, C 0.000 }
gfCNCPoint4[10417] = {X 83.1825, Y 40.9459, Z -5.5000, A 0.000, B 0.000, C 0.000 }
gfCNCPoint4[10418] = {X 83.1823, Y 28.5914, Z -5.5000, A 0.000, B 0.000, C 0.000 }
gfCNCPoint4[10419] = {X 79.1823, Y 28.5914, Z -5.5000, A 0.000, B 0.000, C 0.000 }
gfCNCPoint4[10420] = {X 83.2623, Y 28.5914, Z -5.5000, A 0.000, B 0.000, C 0.000 }
gfCNCPoint4[10421] = {X 83.2622, Y 16.1988, Z -5.5000, A 0.000, B 0.000, C 0.000 }
gfCNCPoint4[10422] = {X 82.6247, Y 15.5491, Z -5.5000, A 0.000, B 0.000, C 0.000 }
gfCNCPoint4[10423] = {X 82.1439, Y 14.7763, Z -5.5000, A 0.000, B 0.000, C 0.000 }
gfCNCPoint4[10424] = {X 81.8425, Y 13.9175, Z -5.5000, A 0.000, B 0.000, C 0.000 }
gfCNCPoint4[10425] = {X 81.7352, Y 13.0136, Z -5.5000, A 0.000, B 0.000, C 0.000 }
gfCNCPoint4[10426] = {X 81.7351, Y 12.1868, Z -5.5000, A 0.000, B 0.000, C 0.000 }
gfCNCPoint4[10427] = {X 81.8394, Y 11.2611, Z -5.5000, A 0.000, B 0.000, C 0.000 }
gfCNCPoint4[10428] = {X 82.1470, Y 10.3819, Z -5.5000, A 0.000, B 0.000, C 0.000 }
gfCNCPoint4[10429] = {X 82.6427, Y 9.5931, Z -5.5000, A 0.000, B 0.000, C 0.000 }
gfCNCPoint4[10430] = {X 83.3014, Y 8.9344, Z -5.5000, A 0.000, B 0.000, C 0.000 }
gfCNCPoint4[10431] = {X 84.0901, Y 8.4388, Z -5.5000, A 0.000, B 0.000, C 0.000 }
gfCNCPoint4[10432] = {X 84.9694, Y 8.1311, Z -5.5000, A 0.000, B 0.000, C 0.000 }
gfCNCPoint4[10433] = {X 85.8951, Y 8.0268, Z -5.5000, A 0.000, B 0.000, C 0.000 }
gfCNCPoint4[10434] = {X 94.0497, Y 8.0268, Z -5.5000, A 0.000, B 0.000, C 0.000 }
gfCNCPoint4[10435] = {X 94.9754, Y 8.1311, Z -5.5000, A 0.000, B 0.000, C 0.000 }
gfCNCPoint4[10436] = {X 95.8546, Y 8.4388, Z -5.5000, A 0.000, B 0.000, C 0.000 }
gfCNCPoint4[10437] = {X 96.6434, Y 8.9344, Z -5.5000, A 0.000, B 0.000, C 0.000 }
gfCNCPoint4[10438] = {X 97.3021, Y 9.5931, Z -5.5000, A 0.000, B 0.000, C 0.000 }
gfCNCPoint4[10439] = {X 97.7977, Y 10.3819, Z -5.5000, A 0.000, B 0.000, C 0.000 }
gfCNCPoint4[10440] = {X 98.1054, Y 11.2611, Z -5.5000, A 0.000, B 0.000, C 0.000 }
gfCNCPoint4[10441] = {X 98.2097, Y 12.1868, Z -5.5000, A 0.000, B 0.000, C 0.000 }
gfCNCPoint4[10442] = {X 98.2097, Y 12.9782, Z -5.5000, A 0.000, B 0.000, C 0.000 }
gfCNCPoint4[10443] = {X 98.1344, Y 13.7658, Z -5.5000, A 0.000, B 0.000, C 0.000 }
gfCNCPoint4[10444] = {X 97.9113, Y 14.5250, Z -5.5000, A 0.000, B 0.000, C 0.000 }
gfCNCPoint4[10445] = {X 97.5485, Y 15.2282, Z -5.5000, A 0.000, B 0.000, C 0.000 }
gfCNCPoint4[10446] = {X 101.8761, Y 25.9517, Z -5.5000, A 0.000, B 0.000, C 0.000 }
gfCNCPoint4[10447] = {X 106.1950, Y 15.2057, Z -5.5000, A 0.000, B 0.000, C 0.000 }
gfCNCPoint4[10448] = {X 105.8447, Y 14.5203, Z -5.5000, A 0.000, B 0.000, C 0.000 }
gfCNCPoint4[10449] = {X 105.6267, Y 13.7821, Z -5.5000, A 0.000, B 0.000, C 0.000 }
gfCNCPoint4[10450] = {X 105.5485, Y 13.0164, Z -5.5000, A 0.000, B 0.000, C 0.000 }
gfCNCPoint4[10451] = {X 105.5483, Y 12.1868, Z -5.5000, A 0.000, B 0.000, C 0.000 }
gfCNCPoint4[10452] = {X 105.6526, Y 11.2611, Z -5.5000, A 0.000, B 0.000, C 0.000 }
gfCNCPoint4[10453] = {X 105.9602, Y 10.3819, Z -5.5000, A 0.000, B 0.000, C 0.000 }
gfCNCPoint4[10454] = {X 106.4559, Y 9.5931, Z -5.5000, A 0.000, B 0.000, C 0.000 }
gfCNCPoint4[10455] = {X 107.1146, Y 8.9344, Z -5.5000, A 0.000, B 0.000, C 0.000 }
gfCNCPoint4[10456] = {X 107.9033, Y 8.4388, Z -5.5000, A 0.000, B 0.000, C 0.000 }
gfCNCPoint4[10457] = {X 108.7826, Y 8.1311, Z -5.5000, A 0.000, B 0.000, C 0.000 }
gfCNCPoint4[10458] = {X 109.7083, Y 8.0268, Z -5.5000, A 0.000, B 0.000, C 0.000 }
gfCNCPoint4[10459] = {X 117.7916, Y 8.0268, Z -5.5000, A 0.000, B 0.000, C 0.000 }
gfCNCPoint4[10460] = {X 118.7173, Y 8.1311, Z -5.5000, A 0.000, B 0.000, C 0.000 }
gfCNCPoint4[10461] = {X 119.5965, Y 8.4388, Z -5.5000, A 0.000, B 0.000, C 0.000 }
gfCNCPoint4[10462] = {X 120.3853, Y 8.9344, Z -5.5000, A 0.000, B 0.000, C 0.000 }
gfCNCPoint4[10463] = {X 121.0440, Y 9.5931, Z -5.5000, A 0.000, B 0.000, C 0.000 }
gfCNCPoint4[10464] = {X 121.5396, Y 10.3819, Z -5.5000, A 0.000, B 0.000, C 0.000 }
gfCNCPoint4[10465] = {X 121.8473, Y 11.2611, Z -5.5000, A 0.000, B 0.000, C 0.000 }
gfCNCPoint4[10466] = {X 121.9516, Y 12.1868, Z -5.5000, A 0.000, B 0.000, C 0.000 }
gfCNCPoint4[10467] = {X 121.9516, Y 12.9782, Z -5.5000, A 0.000, B 0.000, C 0.000 }
gfCNCPoint4[10468] = {X 121.8501, Y 13.8913, Z -5.5000, A 0.000, B 0.000, C 0.000 }
gfCNCPoint4[10469] = {X 121.5506, Y 14.7599, Z -5.5000, A 0.000, B 0.000, C 0.000 }
gfCNCPoint4[10470] = {X 121.0678, Y 15.5416, Z -5.5000, A 0.000, B 0.000, C 0.000 }
gfCNCPoint4[10471] = {X 120.4251, Y 16.1983, Z -5.5000, A 0.000, B 0.000, C 0.000 }
gfCNCPoint4[10472] = {X 120.4244, Y 40.9900, Z -5.5000, A 0.000, B 0.000, C 0.000 }
gfCNCPoint4[10473] = {X 120.5192, Y 41.0679, Z -5.5000, A 0.000, B 0.000, C 0.000 }
gfCNCPoint4[10474] = {X 121.1188, Y 41.7117, Z -5.5000, A 0.000, B 0.000, C 0.000 }
gfCNCPoint4[10475] = {X 121.5695, Y 42.4672, Z -5.5000, A 0.000, B 0.000, C 0.000 }
gfCNCPoint4[10476] = {X 121.8512, Y 43.3007, Z -5.5000, A 0.000, B 0.000, C 0.000 }
gfCNCPoint4[10477] = {X 121.9514, Y 44.1747, Z -5.5000, A 0.000, B 0.000, C 0.000 }
gfCNCPoint4[10478] = {X 121.9516, Y 45.0000, Z -5.5000, A 0.000, B 0.000, C 0.000 }
gfCNCPoint4[10479] = {X 121.8473, Y 45.9257, Z -5.5000, A 0.000, B 0.000, C 0.000 }
gfCNCPoint4[10480] = {X 121.5396, Y 46.8050, Z -5.5000, A 0.000, B 0.000, C 0.000 }
gfCNCPoint4[10481] = {X 121.0440, Y 47.5937, Z -5.5000, A 0.000, B 0.000, C 0.000 }
gfCNCPoint4[10482] = {X 120.3853, Y 48.2524, Z -5.5000, A 0.000, B 0.000, C 0.000 }
gfCNCPoint4[10483] = {X 119.5965, Y 48.7480, Z -5.5000, A 0.000, B 0.000, C 0.000 }
gfCNCPoint4[10484] = {X 118.7173, Y 49.0557, Z -5.5000, A 0.000, B 0.000, C 0.000 }
gfCNCPoint4[10485] = {X 117.7916, Y 49.1600, Z -5.5000, A 0.000, B 0.000, C 0.000 }
gfCNCPoint4[10486] = {X 111.9185, Y 49.1600, Z -5.5000, A 0.000, B 0.000, C 0.000 }
gfCNCPoint4[10487] = {X 110.9974, Y 49.0567, Z -5.5000, A 0.000, B 0.000, C 0.000 }
gfCNCPoint4[10488] = {X 110.1220, Y 48.7521, Z -5.5000, A 0.000, B 0.000, C 0.000 }
gfCNCPoint4[10489] = {X 109.3358, Y 48.2612, Z -5.5000, A 0.000, B 0.000, C 0.000 }
gfCNCPoint4[10490] = {X 108.6778, Y 47.6084, Z -5.5000, A 0.000, B 0.000, C 0.000 }
gfCNCPoint4[10491] = {X 108.1807, Y 46.8261, Z -5.5000, A 0.000, B 0.000, C 0.000 }
gfCNCPoint4[10492] = {X 107.8691, Y 45.9531, Z -5.5000, A 0.000, B 0.000, C 0.000 }
gfCNCPoint4[10493] = {X 107.7586, Y 45.0328, Z -5.5000, A 0.000, B 0.000, C 0.000 }
gfCNCPoint4[10494] = {X 107.7585, Y 44.1807, Z -5.5000, A 0.000, B 0.000, C 0.000 }
gfCNCPoint4[10495] = {X 107.7929, Y 43.6572, Z -5.5000, A 0.000, B 0.000, C 0.000 }
gfCNCPoint4[10496] = {X 107.8955, Y 43.1427, Z -5.5000, A 0.000, B 0.000, C 0.000 }
gfCNCPoint4[10497] = {X 108.0565, Y 42.6653, Z -5.5000, A 0.000, B 0.000, C 0.000 }
gfCNCPoint4[10498] = {X 108.2763, Y 42.2120, Z -5.5000, A 0.000, B 0.000, C 0.000 }
gfCNCPoint4[10499] = {X 108.7345, Y 41.5347, Z -5.5000, A 0.000, B 0.000, C 0.000 }
gfCNCPoint4[10500] = {X 109.2856, Y 40.9305, Z -5.5000, A 0.000, B 0.000, C 0.000 }
gfCNCPoint4[10501] = {X 109.2855, Y 39.0829, Z -5.5000, A 0.000, B 0.000, C 0.000 }
gfCNCPoint4[10502] = {X 109.0402, Y 39.0829, Z -5.5000, A 0.000, B 0.000, C 0.000 }
gfCNCPoint4[10503] = {X 105.9641, Y 46.5999, Z -5.5000, A 0.000, B 0.000, C 0.000 }
gfCNCPoint4[10504] = {X 105.6077, Y 47.2737, Z -5.5000, A 0.000, B 0.000, C 0.000 }
gfCNCPoint4[10505] = {X 105.1344, Y 47.8711, Z -5.5000, A 0.000, B 0.000, C 0.000 }
gfCNCPoint4[10506] = {X 104.5601, Y 48.3721, Z -5.5000, A 0.000, B 0.000, C 0.000 }
gfCNCPoint4[10507] = {X 103.9040, Y 48.7600, Z -5.5000, A 0.000, B 0.000, C 0.000 }
gfCNCPoint4[10508] = {X 102.9952, Y 49.0678, Z -5.5000, A 0.000, B 0.000, C 0.000 }
gfCNCPoint4[10509] = {X 102.0400, Y 49.1592, Z -5.5000, A 0.000, B 0.000, C 0.000 }
gfCNCPoint4[10510] = {X 101.0894, Y 49.0293, Z -5.5000, A 0.000, B 0.000, C 0.000 }
gfCNCPoint4[10511] = {X 100.1937, Y 48.6850, Z -5.5000, A 0.000, B 0.000, C 0.000 }
gfCNCPoint4[10512] = {X 99.4008, Y 48.1448, Z -5.5000, A 0.000, B 0.000, C 0.000 }
gfCNCPoint4[10513] = {X 98.7527, Y 47.4372, Z -5.5000, A 0.000, B 0.000, C 0.000 }
gfCNCPoint4[10514] = {X 98.2840, Y 46.5999, Z -5.5000, A 0.000, B 0.000, C 0.000 }
gfCNCPoint4[10515] = {X 94.9713, Y 38.4983, Z -5.5000, A 0.000, B 0.000, C 0.000 }
gfCNCPoint4[10516] = {X 94.9714, Y 40.9790, Z -5.5000, A 0.000, B 0.000, C 0.000 }
gfCNCPoint4[10517] = {X 95.5112, Y 41.5178, Z -5.5000, A 0.000, B 0.000, C 0.000 }
gfCNCPoint4[10518] = {X 95.9457, Y 42.1445, Z -5.5000, A 0.000, B 0.000, C 0.000 }
gfCNCPoint4[10519] = {X 96.1831, Y 42.6331, Z -5.5000, A 0.000, B 0.000, C 0.000 }
gfCNCPoint4[10520] = {X 96.3561, Y 43.1481, Z -5.5000, A 0.000, B 0.000, C 0.000 }
gfCNCPoint4[10521] = {X 96.4608, Y 43.6734, Z -5.5000, A 0.000, B 0.000, C 0.000 }
gfCNCPoint4[10522] = {X 96.4985, Y 44.2077, Z -5.5000, A 0.000, B 0.000, C 0.000 }
gfCNCPoint4[10523] = {X 96.4983, Y 45.0400, Z -5.5000, A 0.000, B 0.000, C 0.000 }
gfCNCPoint4[10524] = {X 96.3865, Y 45.9591, Z -5.5000, A 0.000, B 0.000, C 0.000 }
gfCNCPoint4[10525] = {X 96.0741, Y 46.8306, Z -5.5000, A 0.000, B 0.000, C 0.000 }
gfCNCPoint4[10526] = {X 95.5767, Y 47.6115, Z -5.5000, A 0.000, B 0.000, C 0.000 }
gfCNCPoint4[10527] = {X 94.9188, Y 48.2631, Z -5.5000, A 0.000, B 0.000, C 0.000 }
gfCNCPoint4[10528] = {X 94.1332, Y 48.7530, Z -5.5000, A 0.000, B 0.000, C 0.000 }
gfCNCPoint4[10529] = {X 93.2587, Y 49.0570, Z -5.5000, A 0.000, B 0.000, C 0.000 }
gfCNCPoint4[10530] = {X 92.3385, Y 49.1600, Z -5.5000, A 0.000, B 0.000, C 0.000 }
gfCNCPoint4[10531] = {X 85.8951, Y 49.1600, Z -5.5000, A 0.000, B 0.000, C 0.000 }
gfCNCPoint4[10532] = {X 84.9741, Y 49.0568, Z -5.5000, A 0.000, B 0.000, C 0.000 }
gfCNCPoint4[10533] = {X 84.0988, Y 48.7522, Z -5.5000, A 0.000, B 0.000, C 0.000 }
gfCNCPoint4[10534] = {X 83.3127, Y 48.2614, Z -5.5000, A 0.000, B 0.000, C 0.000 }
gfCNCPoint4[10535] = {X 82.6547, Y 47.6088, Z -5.5000, A 0.000, B 0.000, C 0.000 }
gfCNCPoint4[10536] = {X 82.1576, Y 46.8267, Z -5.5000, A 0.000, B 0.000, C 0.000 }
gfCNCPoint4[10537] = {X 81.8459, Y 45.9539, Z -5.5000, A 0.000, B 0.000, C 0.000 }
gfCNCPoint4[10538] = {X 81.7352, Y 45.0338, Z -5.5000, A 0.000, B 0.000, C 0.000 }
gfCNCPoint4[10539] = {X 81.7351, Y 44.2080, Z -5.5000, A 0.000, B 0.000, C 0.000 }
gfCNCPoint4[10540] = {X 81.8403, Y 43.2948, Z -5.5000, A 0.000, B 0.000, C 0.000 }
gfCNCPoint4[10541] = {X 82.1409, Y 42.4261, Z -5.5000, A 0.000, B 0.000, C 0.000 }
gfCNCPoint4[10542] = {X 82.6226, Y 41.6432, Z -5.5000, A 0.000, B 0.000, C 0.000 }
gfCNCPoint4[10543] = {X 83.2625, Y 40.9833, Z -5.5000, A 0.000, B 0.000, C 0.000 }
gfCNCPoint4[10544] = {X 83.2623, Y 28.5914, Z -5.5000, A 0.000, B 0.000, C 0.000 }
gfCNCPoint4[10545] = {X 79.2623, Y 28.5914, Z -5.5000, A 0.000, B 0.000, C 0.000 }
gfCNCPoint4[10546] = {X 83.3423, Y 28.5914, Z -5.5000, A 0.000, B 0.000, C 0.000 }
gfCNCPoint4[10547] = {X 83.3422, Y 16.1607, Z -5.5000, A 0.000, B 0.000, C 0.000 }
gfCNCPoint4[10548] = {X 82.7052, Y 15.5219, Z -5.5000, A 0.000, B 0.000, C 0.000 }
gfCNCPoint4[10549] = {X 82.2242, Y 14.7588, Z -5.5000, A 0.000, B 0.000, C 0.000 }
gfCNCPoint4[10550] = {X 81.9226, Y 13.9086, Z -5.5000, A 0.000, B 0.000, C 0.000 }
gfCNCPoint4[10551] = {X 81.8152, Y 13.0129, Z -5.5000, A 0.000, B 0.000, C 0.000 }
gfCNCPoint4[10552] = {X 81.8151, Y 12.1868, Z -5.5000, A 0.000, B 0.000, C 0.000 }
gfCNCPoint4[10553] = {X 81.9174, Y 11.2789, Z -5.5000, A 0.000, B 0.000, C 0.000 }
gfCNCPoint4[10554] = {X 82.2191, Y 10.4166, Z -5.5000, A 0.000, B 0.000, C 0.000 }
gfCNCPoint4[10555] = {X 82.7052, Y 9.6430, Z -5.5000, A 0.000, B 0.000, C 0.000 }
gfCNCPoint4[10556] = {X 83.3512, Y 8.9969, Z -5.5000, A 0.000, B 0.000, C 0.000 }
gfCNCPoint4[10557] = {X 84.1248, Y 8.5109, Z -5.5000, A 0.000, B 0.000, C 0.000 }
gfCNCPoint4[10558] = {X 84.9872, Y 8.2091, Z -5.5000, A 0.000, B 0.000, C 0.000 }
gfCNCPoint4[10559] = {X 85.8951, Y 8.1068, Z -5.5000, A 0.000, B 0.000, C 0.000 }
gfCNCPoint4[10560] = {X 94.0497, Y 8.1068, Z -5.5000, A 0.000, B 0.000, C 0.000 }
gfCNCPoint4[10561] = {X 94.9576, Y 8.2091, Z -5.5000, A 0.000, B 0.000, C 0.000 }
gfCNCPoint4[10562] = {X 95.8199, Y 8.5109, Z -5.5000, A 0.000, B 0.000, C 0.000 }
gfCNCPoint4[10563] = {X 96.5935, Y 8.9969, Z -5.5000, A 0.000, B 0.000, C 0.000 }
gfCNCPoint4[10564] = {X 97.2395, Y 9.6430, Z -5.5000, A 0.000, B 0.000, C 0.000 }
gfCNCPoint4[10565] = {X 97.7256, Y 10.4166, Z -5.5000, A 0.000, B 0.000, C 0.000 }
gfCNCPoint4[10566] = {X 98.0274, Y 11.2789, Z -5.5000, A 0.000, B 0.000, C 0.000 }
gfCNCPoint4[10567] = {X 98.1297, Y 12.1868, Z -5.5000, A 0.000, B 0.000, C 0.000 }
gfCNCPoint4[10568] = {X 98.1297, Y 12.9782, Z -5.5000, A 0.000, B 0.000, C 0.000 }
gfCNCPoint4[10569] = {X 98.0631, Y 13.7119, Z -5.5000, A 0.000, B 0.000, C 0.000 }
gfCNCPoint4[10570] = {X 97.8657, Y 14.4217, Z -5.5000, A 0.000, B 0.000, C 0.000 }
gfCNCPoint4[10571] = {X 97.5439, Y 15.0844, Z -5.5000, A 0.000, B 0.000, C 0.000 }
gfCNCPoint4[10572] = {X 97.4974, Y 15.1596, Z -5.5000, A 0.000, B 0.000, C 0.000 }
gfCNCPoint4[10573] = {X 97.4493, Y 15.2338, Z -5.5000, A 0.000, B 0.000, C 0.000 }
gfCNCPoint4[10574] = {X 97.4857, Y 15.2810, Z -5.5000, A 0.000, B 0.000, C 0.000 }
gfCNCPoint4[10575] = {X 101.8763, Y 26.1659, Z -5.5000, A 0.000, B 0.000, C 0.000 }
gfCNCPoint4[10576] = {X 106.2846, Y 15.1972, Z -5.5000, A 0.000, B 0.000, C 0.000 }
gfCNCPoint4[10577] = {X 106.2411, Y 15.1287, Z -5.5000, A 0.000, B 0.000, C 0.000 }
gfCNCPoint4[10578] = {X 106.1990, Y 15.0593, Z -5.5000, A 0.000, B 0.000, C 0.000 }
gfCNCPoint4[10579] = {X 105.8897, Y 14.4151, Z -5.5000, A 0.000, B 0.000, C 0.000 }
gfCNCPoint4[10580] = {X 105.6976, Y 13.7269, Z -5.5000, A 0.000, B 0.000, C 0.000 }
gfCNCPoint4[10581] = {X 105.6285, Y 13.0157, Z -5.5000, A 0.000, B 0.000, C 0.000 }
gfCNCPoint4[10582] = {X 105.6283, Y 12.1868, Z -5.5000, A 0.000, B 0.000, C 0.000 }
gfCNCPoint4[10583] = {X 105.7306, Y 11.2789, Z -5.5000, A 0.000, B 0.000, C 0.000 }
gfCNCPoint4[10584] = {X 106.0323, Y 10.4166, Z -5.5000, A 0.000, B 0.000, C 0.000 }
gfCNCPoint4[10585] = {X 106.5184, Y 9.6430, Z -5.5000, A 0.000, B 0.000, C 0.000 }
gfCNCPoint4[10586] = {X 107.1644, Y 8.9969, Z -5.5000, A 0.000, B 0.000, C 0.000 }
gfCNCPoint4[10587] = {X 107.9380, Y 8.5109, Z -5.5000, A 0.000, B 0.000, C 0.000 }
gfCNCPoint4[10588] = {X 108.8004, Y 8.2091, Z -5.5000, A 0.000, B 0.000, C 0.000 }
gfCNCPoint4[10589] = {X 109.7083, Y 8.1068, Z -5.5000, A 0.000, B 0.000, C 0.000 }
gfCNCPoint4[10590] = {X 117.7916, Y 8.1068, Z -5.5000, A 0.000, B 0.000, C 0.000 }
gfCNCPoint4[10591] = {X 118.6995, Y 8.2091, Z -5.5000, A 0.000, B 0.000, C 0.000 }
gfCNCPoint4[10592] = {X 119.5618, Y 8.5109, Z -5.5000, A 0.000, B 0.000, C 0.000 }
gfCNCPoint4[10593] = {X 120.3354, Y 8.9969, Z -5.5000, A 0.000, B 0.000, C 0.000 }
gfCNCPoint4[10594] = {X 120.9814, Y 9.6430, Z -5.5000, A 0.000, B 0.000, C 0.000 }
gfCNCPoint4[10595] = {X 121.4675, Y 10.4166, Z -5.5000, A 0.000, B 0.000, C 0.000 }
gfCNCPoint4[10596] = {X 121.7693, Y 11.2789, Z -5.5000, A 0.000, B 0.000, C 0.000 }
gfCNCPoint4[10597] = {X 121.8716, Y 12.1868, Z -5.5000, A 0.000, B 0.000, C 0.000 }
gfCNCPoint4[10598] = {X 121.8716, Y 12.9782, Z -5.5000, A 0.000, B 0.000, C 0.000 }
gfCNCPoint4[10599] = {X 121.7699, Y 13.8830, Z -5.5000, A 0.000, B 0.000, C 0.000 }
gfCNCPoint4[10600] = {X 121.4702, Y 14.7427, Z -5.5000, A 0.000, B 0.000, C 0.000 }
gfCNCPoint4[10601] = {X 120.9872, Y 15.5146, Z -5.5000, A 0.000, B 0.000, C 0.000 }
gfCNCPoint4[10602] = {X 120.3451, Y 16.1601, Z -5.5000, A 0.000, B 0.000, C 0.000 }
gfCNCPoint4[10603] = {X 120.3444, Y 41.0279, Z -5.5000, A 0.000, B 0.000, C 0.000 }
gfCNCPoint4[10604] = {X 120.4676, Y 41.1290, Z -5.5000, A 0.000, B 0.000, C 0.000 }
gfCNCPoint4[10605] = {X 121.0553, Y 41.7604, Z -5.5000, A 0.000, B 0.000, C 0.000 }
gfCNCPoint4[10606] = {X 121.4971, Y 42.5012, Z -5.5000, A 0.000, B 0.000, C 0.000 }
gfCNCPoint4[10607] = {X 121.7732, Y 43.3184, Z -5.5000, A 0.000, B 0.000, C 0.000 }
gfCNCPoint4[10608] = {X 121.8714, Y 44.1754, Z -5.5000, A 0.000, B 0.000, C 0.000 }
gfCNCPoint4[10609] = {X 121.8716, Y 45.0000, Z -5.5000, A 0.000, B 0.000, C 0.000 }
gfCNCPoint4[10610] = {X 121.7693, Y 45.9079, Z -5.5000, A 0.000, B 0.000, C 0.000 }
gfCNCPoint4[10611] = {X 121.4675, Y 46.7702, Z -5.5000, A 0.000, B 0.000, C 0.000 }
gfCNCPoint4[10612] = {X 120.9814, Y 47.5438, Z -5.5000, A 0.000, B 0.000, C 0.000 }
gfCNCPoint4[10613] = {X 120.3354, Y 48.1899, Z -5.5000, A 0.000, B 0.000, C 0.000 }
gfCNCPoint4[10614] = {X 119.5618, Y 48.6760, Z -5.5000, A 0.000, B 0.000, C 0.000 }
gfCNCPoint4[10615] = {X 118.6995, Y 48.9777, Z -5.5000, A 0.000, B 0.000, C 0.000 }
gfCNCPoint4[10616] = {X 117.7916, Y 49.0800, Z -5.5000, A 0.000, B 0.000, C 0.000 }
gfCNCPoint4[10617] = {X 111.9185, Y 49.0800, Z -5.5000, A 0.000, B 0.000, C 0.000 }
gfCNCPoint4[10618] = {X 111.0151, Y 48.9787, Z -5.5000, A 0.000, B 0.000, C 0.000 }
gfCNCPoint4[10619] = {X 110.1565, Y 48.6799, Z -5.5000, A 0.000, B 0.000, C 0.000 }
gfCNCPoint4[10620] = {X 109.3855, Y 48.1985, Z -5.5000, A 0.000, B 0.000, C 0.000 }
gfCNCPoint4[10621] = {X 108.7401, Y 47.5582, Z -5.5000, A 0.000, B 0.000, C 0.000 }
gfCNCPoint4[10622] = {X 108.2526, Y 46.7909, Z -5.5000, A 0.000, B 0.000, C 0.000 }
gfCNCPoint4[10623] = {X 107.9470, Y 45.9348, Z -5.5000, A 0.000, B 0.000, C 0.000 }
gfCNCPoint4[10624] = {X 107.8386, Y 45.0322, Z -5.5000, A 0.000, B 0.000, C 0.000 }
gfCNCPoint4[10625] = {X 107.8385, Y 44.1807, Z -5.5000, A 0.000, B 0.000, C 0.000 }
gfCNCPoint4[10626] = {X 107.8722, Y 43.6677, Z -5.5000, A 0.000, B 0.000, C 0.000 }
gfCNCPoint4[10627] = {X 107.9727, Y 43.1635, Z -5.5000, A 0.000, B 0.000, C 0.000 }
gfCNCPoint4[10628] = {X 108.1306, Y 42.6956, Z -5.5000, A 0.000, B 0.000, C 0.000 }
gfCNCPoint4[10629] = {X 108.3460, Y 42.2513, Z -5.5000, A 0.000, B 0.000, C 0.000 }
gfCNCPoint4[10630] = {X 108.8082, Y 41.5704, Z -5.5000, A 0.000, B 0.000, C 0.000 }
gfCNCPoint4[10631] = {X 109.3656, Y 40.9650, Z -5.5000, A 0.000, B 0.000, C 0.000 }
gfCNCPoint4[10632] = {X 109.3655, Y 39.0029, Z -5.5000, A 0.000, B 0.000, C 0.000 }
gfCNCPoint4[10633] = {X 108.9865, Y 39.0029, Z -5.5000, A 0.000, B 0.000, C 0.000 }
gfCNCPoint4[10634] = {X 105.8902, Y 46.5692, Z -5.5000, A 0.000, B 0.000, C 0.000 }
gfCNCPoint4[10635] = {X 105.5407, Y 47.2300, Z -5.5000, A 0.000, B 0.000, C 0.000 }
gfCNCPoint4[10636] = {X 105.0765, Y 47.8159, Z -5.5000, A 0.000, B 0.000, C 0.000 }
gfCNCPoint4[10637] = {X 104.5133, Y 48.3073, Z -5.5000, A 0.000, B 0.000, C 0.000 }
gfCNCPoint4[10638] = {X 103.8698, Y 48.6877, Z -5.5000, A 0.000, B 0.000, C 0.000 }
gfCNCPoint4[10639] = {X 102.9784, Y 48.9895, Z -5.5000, A 0.000, B 0.000, C 0.000 }
gfCNCPoint4[10640] = {X 102.0417, Y 49.0792, Z -5.5000, A 0.000, B 0.000, C 0.000 }
gfCNCPoint4[10641] = {X 101.1093, Y 48.9518, Z -5.5000, A 0.000, B 0.000, C 0.000 }
gfCNCPoint4[10642] = {X 100.2309, Y 48.6142, Z -5.5000, A 0.000, B 0.000, C 0.000 }
gfCNCPoint4[10643] = {X 99.4532, Y 48.0843, Z -5.5000, A 0.000, B 0.000, C 0.000 }
gfCNCPoint4[10644] = {X 98.8176, Y 47.3903, Z -5.5000, A 0.000, B 0.000, C 0.000 }
gfCNCPoint4[10645] = {X 98.3579, Y 46.5692, Z -5.5000, A 0.000, B 0.000, C 0.000 }
gfCNCPoint4[10646] = {X 94.8923, Y 38.0938, Z -5.5000, A 0.000, B 0.000, C 0.000 }
gfCNCPoint4[10647] = {X 94.8913, Y 38.2309, Z -5.5000, A 0.000, B 0.000, C 0.000 }
gfCNCPoint4[10648] = {X 94.8914, Y 41.0167, Z -5.5000, A 0.000, B 0.000, C 0.000 }
gfCNCPoint4[10649] = {X 95.4378, Y 41.5548, Z -5.5000, A 0.000, B 0.000, C 0.000 }
gfCNCPoint4[10650] = {X 95.8762, Y 42.1840, Z -5.5000, A 0.000, B 0.000, C 0.000 }
gfCNCPoint4[10651] = {X 96.1090, Y 42.6634, Z -5.5000, A 0.000, B 0.000, C 0.000 }
gfCNCPoint4[10652] = {X 96.2788, Y 43.1686, Z -5.5000, A 0.000, B 0.000, C 0.000 }
gfCNCPoint4[10653] = {X 96.3815, Y 43.6840, Z -5.5000, A 0.000, B 0.000, C 0.000 }
gfCNCPoint4[10654] = {X 96.4185, Y 44.2083, Z -5.5000, A 0.000, B 0.000, C 0.000 }
gfCNCPoint4[10655] = {X 96.4184, Y 45.0392, Z -5.5000, A 0.000, B 0.000, C 0.000 }
gfCNCPoint4[10656] = {X 96.3086, Y 45.9406, Z -5.5000, A 0.000, B 0.000, C 0.000 }
gfCNCPoint4[10657] = {X 96.0023, Y 46.7954, Z -5.5000, A 0.000, B 0.000, C 0.000 }
gfCNCPoint4[10658] = {X 95.5144, Y 47.5613, Z -5.5000, A 0.000, B 0.000, C 0.000 }
gfCNCPoint4[10659] = {X 94.8692, Y 48.2003, Z -5.5000, A 0.000, B 0.000, C 0.000 }
gfCNCPoint4[10660] = {X 94.0987, Y 48.6808, Z -5.5000, A 0.000, B 0.000, C 0.000 }
gfCNCPoint4[10661] = {X 93.2410, Y 48.9789, Z -5.5000, A 0.000, B 0.000, C 0.000 }
gfCNCPoint4[10662] = {X 92.3385, Y 49.0800, Z -5.5000, A 0.000, B 0.000, C 0.000 }
gfCNCPoint4[10663] = {X 85.8951, Y 49.0800, Z -5.5000, A 0.000, B 0.000, C 0.000 }
gfCNCPoint4[10664] = {X 84.9918, Y 48.9788, Z -5.5000, A 0.000, B 0.000, C 0.000 }
gfCNCPoint4[10665] = {X 84.1334, Y 48.6801, Z -5.5000, A 0.000, B 0.000, C 0.000 }
gfCNCPoint4[10666] = {X 83.3624, Y 48.1987, Z -5.5000, A 0.000, B 0.000, C 0.000 }
gfCNCPoint4[10667] = {X 82.7171, Y 47.5586, Z -5.5000, A 0.000, B 0.000, C 0.000 }
gfCNCPoint4[10668] = {X 82.2295, Y 46.7916, Z -5.5000, A 0.000, B 0.000, C 0.000 }
gfCNCPoint4[10669] = {X 81.9238, Y 45.9356, Z -5.5000, A 0.000, B 0.000, C 0.000 }
gfCNCPoint4[10670] = {X 81.8152, Y 45.0332, Z -5.5000, A 0.000, B 0.000, C 0.000 }
gfCNCPoint4[10671] = {X 81.8151, Y 44.2084, Z -5.5000, A 0.000, B 0.000, C 0.000 }
gfCNCPoint4[10672] = {X 81.9204, Y 43.3034, Z -5.5000, A 0.000, B 0.000, C 0.000 }
gfCNCPoint4[10673] = {X 82.2213, Y 42.4435, Z -5.5000, A 0.000, B 0.000, C 0.000 }
gfCNCPoint4[10674] = {X 82.7031, Y 41.6702, Z -5.5000, A 0.000, B 0.000, C 0.000 }
gfCNCPoint4[10675] = {X 83.3425, Y 41.0211, Z -5.5000, A 0.000, B 0.000, C 0.000 }
gfCNCPoint4[10676] = {X 83.3423, Y 28.5914, Z -5.5000, A 0.000, B 0.000, C 0.000 }
gfCNCPoint4[10677] = {X 79.3423, Y 28.5914, Z -5.5000, A 0.000, B 0.000, C 0.000 }
gfCNCPoint4[10678] = {X 83.4223, Y 28.5914, Z -5.5000, A 0.000, B 0.000, C 0.000 }
gfCNCPoint4[10679] = {X 83.4222, Y 16.1220, Z -5.5000, A 0.000, B 0.000, C 0.000 }
gfCNCPoint4[10680] = {X 82.7804, Y 15.4877, Z -5.5000, A 0.000, B 0.000, C 0.000 }
gfCNCPoint4[10681] = {X 82.2970, Y 14.7256, Z -5.5000, A 0.000, B 0.000, C 0.000 }
gfCNCPoint4[10682] = {X 81.9969, Y 13.8746, Z -5.5000, A 0.000, B 0.000, C 0.000 }
gfCNCPoint4[10683] = {X 81.8951, Y 12.9780, Z -5.5000, A 0.000, B 0.000, C 0.000 }
gfCNCPoint4[10684] = {X 81.8951, Y 12.1868, Z -5.5000, A 0.000, B 0.000, C 0.000 }
gfCNCPoint4[10685] = {X 81.9954, Y 11.2967, Z -5.5000, A 0.000, B 0.000, C 0.000 }
gfCNCPoint4[10686] = {X 82.2912, Y 10.4513, Z -5.5000, A 0.000, B 0.000, C 0.000 }
gfCNCPoint4[10687] = {X 82.7677, Y 9.6929, Z -5.5000, A 0.000, B 0.000, C 0.000 }
gfCNCPoint4[10688] = {X 83.4011, Y 9.0595, Z -5.5000, A 0.000, B 0.000, C 0.000 }
gfCNCPoint4[10689] = {X 84.1595, Y 8.5829, Z -5.5000, A 0.000, B 0.000, C 0.000 }
gfCNCPoint4[10690] = {X 85.0050, Y 8.2871, Z -5.5000, A 0.000, B 0.000, C 0.000 }
gfCNCPoint4[10691] = {X 85.8951, Y 8.1868, Z -5.5000, A 0.000, B 0.000, C 0.000 }
gfCNCPoint4[10692] = {X 94.0497, Y 8.1868, Z -5.5000, A 0.000, B 0.000, C 0.000 }
gfCNCPoint4[10693] = {X 94.9398, Y 8.2871, Z -5.5000, A 0.000, B 0.000, C 0.000 }
gfCNCPoint4[10694] = {X 95.7852, Y 8.5829, Z -5.5000, A 0.000, B 0.000, C 0.000 }
gfCNCPoint4[10695] = {X 96.5436, Y 9.0595, Z -5.5000, A 0.000, B 0.000, C 0.000 }
gfCNCPoint4[10696] = {X 97.1770, Y 9.6929, Z -5.5000, A 0.000, B 0.000, C 0.000 }
gfCNCPoint4[10697] = {X 97.6535, Y 10.4513, Z -5.5000, A 0.000, B 0.000, C 0.000 }
gfCNCPoint4[10698] = {X 97.9494, Y 11.2967, Z -5.5000, A 0.000, B 0.000, C 0.000 }
gfCNCPoint4[10699] = {X 98.0497, Y 12.1868, Z -5.5000, A 0.000, B 0.000, C 0.000 }
gfCNCPoint4[10700] = {X 98.0495, Y 13.0192, Z -5.5000, A 0.000, B 0.000, C 0.000 }
gfCNCPoint4[10701] = {X 97.9794, Y 13.7244, Z -5.5000, A 0.000, B 0.000, C 0.000 }
gfCNCPoint4[10702] = {X 97.7860, Y 14.4061, Z -5.5000, A 0.000, B 0.000, C 0.000 }
gfCNCPoint4[10703] = {X 97.4754, Y 15.0431, Z -5.5000, A 0.000, B 0.000, C 0.000 }
gfCNCPoint4[10704] = {X 97.4130, Y 15.1433, Z -5.5000, A 0.000, B 0.000, C 0.000 }
gfCNCPoint4[10705] = {X 97.3476, Y 15.2415, Z -5.5000, A 0.000, B 0.000, C 0.000 }
gfCNCPoint4[10706] = {X 97.4115, Y 15.3108, Z -5.5000, A 0.000, B 0.000, C 0.000 }
gfCNCPoint4[10707] = {X 97.9971, Y 16.7687, Z -5.5000, A 0.000, B 0.000, C 0.000 }
gfCNCPoint4[10708] = {X 101.6279, Y 25.7689, Z -5.5000, A 0.000, B 0.000, C 0.000 }
gfCNCPoint4[10709] = {X 101.8768, Y 26.3791, Z -5.5000, A 0.000, B 0.000, C 0.000 }
gfCNCPoint4[10710] = {X 103.7914, Y 21.6150, Z -5.5000, A 0.000, B 0.000, C 0.000 }
gfCNCPoint4[10711] = {X 106.3416, Y 15.2554, Z -5.5000, A 0.000, B 0.000, C 0.000 }
gfCNCPoint4[10712] = {X 106.3813, Y 15.1986, Z -5.5000, A 0.000, B 0.000, C 0.000 }
gfCNCPoint4[10713] = {X 106.3234, Y 15.1093, Z -5.5000, A 0.000, B 0.000, C 0.000 }
gfCNCPoint4[10714] = {X 106.2678, Y 15.0185, Z -5.5000, A 0.000, B 0.000, C 0.000 }
gfCNCPoint4[10715] = {X 105.9603, Y 14.3754, Z -5.5000, A 0.000, B 0.000, C 0.000 }
gfCNCPoint4[10716] = {X 105.7718, Y 13.6879, Z -5.5000, A 0.000, B 0.000, C 0.000 }
gfCNCPoint4[10717] = {X 105.7083, Y 12.9779, Z -5.5000, A 0.000, B 0.000, C 0.000 }
gfCNCPoint4[10718] = {X 105.7083, Y 12.1868, Z -5.5000, A 0.000, B 0.000, C 0.000 }
gfCNCPoint4[10719] = {X 105.8086, Y 11.2967, Z -5.5000, A 0.000, B 0.000, C 0.000 }
gfCNCPoint4[10720] = {X 106.1044, Y 10.4513, Z -5.5000, A 0.000, B 0.000, C 0.000 }
gfCNCPoint4[10721] = {X 106.5810, Y 9.6929, Z -5.5000, A 0.000, B 0.000, C 0.000 }
gfCNCPoint4[10722] = {X 107.2143, Y 9.0595, Z -5.5000, A 0.000, B 0.000, C 0.000 }
gfCNCPoint4[10723] = {X 107.9727, Y 8.5829, Z -5.5000, A 0.000, B 0.000, C 0.000 }
gfCNCPoint4[10724] = {X 108.8182, Y 8.2871, Z -5.5000, A 0.000, B 0.000, C 0.000 }
gfCNCPoint4[10725] = {X 109.7083, Y 8.1868, Z -5.5000, A 0.000, B 0.000, C 0.000 }
gfCNCPoint4[10726] = {X 117.7916, Y 8.1868, Z -5.5000, A 0.000, B 0.000, C 0.000 }
gfCNCPoint4[10727] = {X 118.6817, Y 8.2871, Z -5.5000, A 0.000, B 0.000, C 0.000 }
gfCNCPoint4[10728] = {X 119.5271, Y 8.5829, Z -5.5000, A 0.000, B 0.000, C 0.000 }
gfCNCPoint4[10729] = {X 120.2855, Y 9.0595, Z -5.5000, A 0.000, B 0.000, C 0.000 }
gfCNCPoint4[10730] = {X 120.9189, Y 9.6929, Z -5.5000, A 0.000, B 0.000, C 0.000 }
gfCNCPoint4[10731] = {X 121.3955, Y 10.4513, Z -5.5000, A 0.000, B 0.000, C 0.000 }
gfCNCPoint4[10732] = {X 121.6913, Y 11.2967, Z -5.5000, A 0.000, B 0.000, C 0.000 }
gfCNCPoint4[10733] = {X 121.7916, Y 12.1868, Z -5.5000, A 0.000, B 0.000, C 0.000 }
gfCNCPoint4[10734] = {X 121.7914, Y 13.0192, Z -5.5000, A 0.000, B 0.000, C 0.000 }
gfCNCPoint4[10735] = {X 121.6828, Y 13.9045, Z -5.5000, A 0.000, B 0.000, C 0.000 }
gfCNCPoint4[10736] = {X 121.3807, Y 14.7438, Z -5.5000, A 0.000, B 0.000, C 0.000 }
gfCNCPoint4[10737] = {X 120.9002, Y 15.4952, Z -5.5000, A 0.000, B 0.000, C 0.000 }
gfCNCPoint4[10738] = {X 120.2651, Y 16.1215, Z -5.5000, A 0.000, B 0.000, C 0.000 }
gfCNCPoint4[10739] = {X 120.2644, Y 41.0657, Z -5.5000, A 0.000, B 0.000, C 0.000 }
gfCNCPoint4[10740] = {X 120.4160, Y 41.1901, Z -5.5000, A 0.000, B 0.000, C 0.000 }
gfCNCPoint4[10741] = {X 120.9967, Y 41.8157, Z -5.5000, A 0.000, B 0.000, C 0.000 }
gfCNCPoint4[10742] = {X 121.4315, Y 42.5502, Z -5.5000, A 0.000, B 0.000, C 0.000 }
gfCNCPoint4[10743] = {X 121.7005, Y 43.3602, Z -5.5000, A 0.000, B 0.000, C 0.000 }
gfCNCPoint4[10744] = {X 121.7916, Y 44.2089, Z -5.5000, A 0.000, B 0.000, C 0.000 }
gfCNCPoint4[10745] = {X 121.7916, Y 45.0000, Z -5.5000, A 0.000, B 0.000, C 0.000 }
gfCNCPoint4[10746] = {X 121.6913, Y 45.8901, Z -5.5000, A 0.000, B 0.000, C 0.000 }
gfCNCPoint4[10747] = {X 121.3955, Y 46.7355, Z -5.5000, A 0.000, B 0.000, C 0.000 }
gfCNCPoint4[10748] = {X 120.9189, Y 47.4940, Z -5.5000, A 0.000, B 0.000, C 0.000 }
gfCNCPoint4[10749] = {X 120.2855, Y 48.1273, Z -5.5000, A 0.000, B 0.000, C 0.000 }
gfCNCPoint4[10750] = {X 119.5271, Y 48.6039, Z -5.5000, A 0.000, B 0.000, C 0.000 }
gfCNCPoint4[10751] = {X 118.6817, Y 48.8997, Z -5.5000, A 0.000, B 0.000, C 0.000 }
gfCNCPoint4[10752] = {X 117.7916, Y 49.0000, Z -5.5000, A 0.000, B 0.000, C 0.000 }
gfCNCPoint4[10753] = {X 111.9185, Y 49.0000, Z -5.5000, A 0.000, B 0.000, C 0.000 }
gfCNCPoint4[10754] = {X 111.0284, Y 48.8997, Z -5.5000, A 0.000, B 0.000, C 0.000 }
gfCNCPoint4[10755] = {X 110.1829, Y 48.6039, Z -5.5000, A 0.000, B 0.000, C 0.000 }
gfCNCPoint4[10756] = {X 109.4245, Y 48.1273, Z -5.5000, A 0.000, B 0.000, C 0.000 }
gfCNCPoint4[10757] = {X 108.7911, Y 47.4939, Z -5.5000, A 0.000, B 0.000, C 0.000 }
gfCNCPoint4[10758] = {X 108.3146, Y 46.7355, Z -5.5000, A 0.000, B 0.000, C 0.000 }
gfCNCPoint4[10759] = {X 108.0188, Y 45.8901, Z -5.5000, A 0.000, B 0.000, C 0.000 }
gfCNCPoint4[10760] = {X 107.9185, Y 45.0000, Z -5.5000, A 0.000, B 0.000, C 0.000 }
gfCNCPoint4[10761] = {X 107.9185, Y 44.1807, Z -5.5000, A 0.000, B 0.000, C 0.000 }
gfCNCPoint4[10762] = {X 107.9515, Y 43.6782, Z -5.5000, A 0.000, B 0.000, C 0.000 }
gfCNCPoint4[10763] = {X 108.0500, Y 43.1842, Z -5.5000, A 0.000, B 0.000, C 0.000 }
gfCNCPoint4[10764] = {X 108.2046, Y 42.7259, Z -5.5000, A 0.000, B 0.000, C 0.000 }
gfCNCPoint4[10765] = {X 108.4156, Y 42.2907, Z -5.5000, A 0.000, B 0.000, C 0.000 }
gfCNCPoint4[10766] = {X 108.4427, Y 42.2436, Z -5.5000, A 0.000, B 0.000, C 0.000 }
gfCNCPoint4[10767] = {X 108.4704, Y 42.1970, Z -5.5000, A 0.000, B 0.000, C 0.000 }
gfCNCPoint4[10768] = {X 108.9157, Y 41.5640, Z -5.5000, A 0.000, B 0.000, C 0.000 }
gfCNCPoint4[10769] = {X 109.4456, Y 40.9999, Z -5.5000, A 0.000, B 0.000, C 0.000 }
gfCNCPoint4[10770] = {X 109.4455, Y 38.9229, Z -5.5000, A 0.000, B 0.000, C 0.000 }
gfCNCPoint4[10771] = {X 108.9328, Y 38.9229, Z -5.5000, A 0.000, B 0.000, C 0.000 }
gfCNCPoint4[10772] = {X 105.8164, Y 46.5384, Z -5.5000, A 0.000, B 0.000, C 0.000 }
gfCNCPoint4[10773] = {X 105.3339, Y 47.3869, Z -5.5000, A 0.000, B 0.000, C 0.000 }
gfCNCPoint4[10774] = {X 104.6602, Y 48.0932, Z -5.5000, A 0.000, B 0.000, C 0.000 }
gfCNCPoint4[10775] = {X 103.8355, Y 48.6154, Z -5.5000, A 0.000, B 0.000, C 0.000 }
gfCNCPoint4[10776] = {X 102.9580, Y 48.9121, Z -5.5000, A 0.000, B 0.000, C 0.000 }
gfCNCPoint4[10777] = {X 102.0357, Y 48.9990, Z -5.5000, A 0.000, B 0.000, C 0.000 }
gfCNCPoint4[10778] = {X 101.1182, Y 48.8715, Z -5.5000, A 0.000, B 0.000, C 0.000 }
gfCNCPoint4[10779] = {X 100.2546, Y 48.5362, Z -5.5000, A 0.000, B 0.000, C 0.000 }
gfCNCPoint4[10780] = {X 99.4912, Y 48.0114, Z -5.5000, A 0.000, B 0.000, C 0.000 }
gfCNCPoint4[10781] = {X 98.8691, Y 47.3250, Z -5.5000, A 0.000, B 0.000, C 0.000 }
gfCNCPoint4[10782] = {X 98.4216, Y 46.5139, Z -5.5000, A 0.000, B 0.000, C 0.000 }
gfCNCPoint4[10783] = {X 94.8154, Y 37.6942, Z -5.5000, A 0.000, B 0.000, C 0.000 }
gfCNCPoint4[10784] = {X 94.8113, Y 38.2306, Z -5.5000, A 0.000, B 0.000, C 0.000 }
gfCNCPoint4[10785] = {X 94.8114, Y 41.0549, Z -5.5000, A 0.000, B 0.000, C 0.000 }
gfCNCPoint4[10786] = {X 95.3644, Y 41.5920, Z -5.5000, A 0.000, B 0.000, C 0.000 }
gfCNCPoint4[10787] = {X 95.8066, Y 42.2235, Z -5.5000, A 0.000, B 0.000, C 0.000 }
gfCNCPoint4[10788] = {X 96.0350, Y 42.6937, Z -5.5000, A 0.000, B 0.000, C 0.000 }
gfCNCPoint4[10789] = {X 96.2014, Y 43.1892, Z -5.5000, A 0.000, B 0.000, C 0.000 }
gfCNCPoint4[10790] = {X 96.3022, Y 43.6947, Z -5.5000, A 0.000, B 0.000, C 0.000 }
gfCNCPoint4[10791] = {X 96.3385, Y 44.2089, Z -5.5000, A 0.000, B 0.000, C 0.000 }
gfCNCPoint4[10792] = {X 96.3384, Y 45.0384, Z -5.5000, A 0.000, B 0.000, C 0.000 }
gfCNCPoint4[10793] = {X 96.2308, Y 45.9222, Z -5.5000, A 0.000, B 0.000, C 0.000 }
gfCNCPoint4[10794] = {X 95.9304, Y 46.7602, Z -5.5000, A 0.000, B 0.000, C 0.000 }
gfCNCPoint4[10795] = {X 95.4521, Y 47.5111, Z -5.5000, A 0.000, B 0.000, C 0.000 }
gfCNCPoint4[10796] = {X 94.8196, Y 48.1376, Z -5.5000, A 0.000, B 0.000, C 0.000 }
gfCNCPoint4[10797] = {X 94.0642, Y 48.6086, Z -5.5000, A 0.000, B 0.000, C 0.000 }
gfCNCPoint4[10798] = {X 93.2233, Y 48.9009, Z -5.5000, A 0.000, B 0.000, C 0.000 }
gfCNCPoint4[10799] = {X 92.3385, Y 49.0000, Z -5.5000, A 0.000, B 0.000, C 0.000 }
gfCNCPoint4[10800] = {X 85.8951, Y 49.0000, Z -5.5000, A 0.000, B 0.000, C 0.000 }
gfCNCPoint4[10801] = {X 85.0050, Y 48.8997, Z -5.5000, A 0.000, B 0.000, C 0.000 }
gfCNCPoint4[10802] = {X 84.1595, Y 48.6039, Z -5.5000, A 0.000, B 0.000, C 0.000 }
gfCNCPoint4[10803] = {X 83.4011, Y 48.1273, Z -5.5000, A 0.000, B 0.000, C 0.000 }
gfCNCPoint4[10804] = {X 82.7677, Y 47.4939, Z -5.5000, A 0.000, B 0.000, C 0.000 }
gfCNCPoint4[10805] = {X 82.2912, Y 46.7355, Z -5.5000, A 0.000, B 0.000, C 0.000 }
gfCNCPoint4[10806] = {X 81.9954, Y 45.8901, Z -5.5000, A 0.000, B 0.000, C 0.000 }
gfCNCPoint4[10807] = {X 81.8951, Y 45.0000, Z -5.5000, A 0.000, B 0.000, C 0.000 }
gfCNCPoint4[10808] = {X 81.8951, Y 44.2089, Z -5.5000, A 0.000, B 0.000, C 0.000 }
gfCNCPoint4[10809] = {X 82.0005, Y 43.3121, Z -5.5000, A 0.000, B 0.000, C 0.000 }
gfCNCPoint4[10810] = {X 82.3017, Y 42.4609, Z -5.5000, A 0.000, B 0.000, C 0.000 }
gfCNCPoint4[10811] = {X 82.7836, Y 41.6974, Z -5.5000, A 0.000, B 0.000, C 0.000 }
gfCNCPoint4[10812] = {X 83.4225, Y 41.0594, Z -5.5000, A 0.000, B 0.000, C 0.000 }
gfCNCPoint4[10813] = {X 83.4223, Y 28.5914, Z -5.5000, A 0.000, B 0.000, C 0.000 }
gfCNCPoint4[10814] = {X 79.3423, Y 28.5914, Z -5.5000, A 0.000, B 0.000, C 0.000 }
gfCNCPoint4[10815] = {X 79.3423, Y 28.5914, Z -2.5000, A 0.000, B 0.000, C 0.000 }
gfCNCPoint4[10816] = {X 79.3423, Y 28.5914, Z 11.0000, A 0.000, B 0.000, C 0.000 }
gfCNCPoint4[10817] = {X 136.1636, Y 30.3967, Z 11.0000, A 0.000, B 0.000, C 0.000 }
gfCNCPoint4[10818] = {X 136.1636, Y 30.3967, Z -2.5000, A 0.000, B 0.000, C 0.000 }
gfCNCPoint4[10819] = {X 136.1636, Y 30.3967, Z -5.5000, A 0.000, B 0.000, C 0.000 }
gfCNCPoint4[10820] = {X 140.2436, Y 30.3967, Z -5.5000, A 0.000, B 0.000, C 0.000 }
gfCNCPoint4[10821] = {X 140.2436, Y 19.8777, Z -5.5000, A 0.000, B 0.000, C 0.000 }
gfCNCPoint4[10822] = {X 137.4238, Y 19.8772, Z -5.5000, A 0.000, B 0.000, C 0.000 }
gfCNCPoint4[10823] = {X 136.8914, Y 20.5219, Z -5.5000, A 0.000, B 0.000, C 0.000 }
gfCNCPoint4[10824] = {X 136.2448, Y 21.0519, Z -5.5000, A 0.000, B 0.000, C 0.000 }
gfCNCPoint4[10825] = {X 135.5082, Y 21.4474, Z -5.5000, A 0.000, B 0.000, C 0.000 }
gfCNCPoint4[10826] = {X 134.7093, Y 21.6937, Z -5.5000, A 0.000, B 0.000, C 0.000 }
gfCNCPoint4[10827] = {X 133.8778, Y 21.7814, Z -5.5000, A 0.000, B 0.000, C 0.000 }
gfCNCPoint4[10828] = {X 133.2006, Y 21.7815, Z -5.5000, A 0.000, B 0.000, C 0.000 }
gfCNCPoint4[10829] = {X 132.2394, Y 21.6732, Z -5.5000, A 0.000, B 0.000, C 0.000 }
gfCNCPoint4[10830] = {X 131.3263, Y 21.3537, Z -5.5000, A 0.000, B 0.000, C 0.000 }
gfCNCPoint4[10831] = {X 130.5072, Y 20.8390, Z -5.5000, A 0.000, B 0.000, C 0.000 }
gfCNCPoint4[10832] = {X 129.8231, Y 20.1550, Z -5.5000, A 0.000, B 0.000, C 0.000 }
gfCNCPoint4[10833] = {X 129.3085, Y 19.3359, Z -5.5000, A 0.000, B 0.000, C 0.000 }
gfCNCPoint4[10834] = {X 128.9890, Y 18.4228, Z -5.5000, A 0.000, B 0.000, C 0.000 }
gfCNCPoint4[10835] = {X 128.8806, Y 17.4615, Z -5.5000, A 0.000, B 0.000, C 0.000 }
gfCNCPoint4[10836] = {X 128.8806, Y 10.4835, Z -5.5000, A 0.000, B 0.000, C 0.000 }
gfCNCPoint4[10837] = {X 128.9874, Y 9.5289, Z -5.5000, A 0.000, B 0.000, C 0.000 }
gfCNCPoint4[10838] = {X 129.3026, Y 8.6214, Z -5.5000, A 0.000, B 0.000, C 0.000 }
gfCNCPoint4[10839] = {X 129.8104, Y 7.8061, Z -5.5000, A 0.000, B 0.000, C 0.000 }
gfCNCPoint4[10840] = {X 130.4859, Y 7.1231, Z -5.5000, A 0.000, B 0.000, C 0.000 }
gfCNCPoint4[10841] = {X 131.2956, Y 6.6063, Z -5.5000, A 0.000, B 0.000, C 0.000 }
gfCNCPoint4[10842] = {X 132.1995, Y 6.2811, Z -5.5000, A 0.000, B 0.000, C 0.000 }
gfCNCPoint4[10843] = {X 133.1529, Y 6.1638, Z -5.5000, A 0.000, B 0.000, C 0.000 }
gfCNCPoint4[10844] = {X 133.8866, Y 6.1637, Z -5.5000, A 0.000, B 0.000, C 0.000 }
gfCNCPoint4[10845] = {X 134.7110, Y 6.2518, Z -5.5000, A 0.000, B 0.000, C 0.000 }
gfCNCPoint4[10846] = {X 135.5034, Y 6.4956, Z -5.5000, A 0.000, B 0.000, C 0.000 }
gfCNCPoint4[10847] = {X 136.2346, Y 6.8864, Z -5.5000, A 0.000, B 0.000, C 0.000 }
gfCNCPoint4[10848] = {X 136.8777, Y 7.4096, Z -5.5000, A 0.000, B 0.000, C 0.000 }
gfCNCPoint4[10849] = {X 137.4090, Y 8.0460, Z -5.5000, A 0.000, B 0.000, C 0.000 }
gfCNCPoint4[10850] = {X 155.1129, Y 8.0473, Z -5.5000, A 0.000, B 0.000, C 0.000 }
gfCNCPoint4[10851] = {X 155.6449, Y 7.4097, Z -5.5000, A 0.000, B 0.000, C 0.000 }
gfCNCPoint4[10852] = {X 156.2891, Y 6.8857, Z -5.5000, A 0.000, B 0.000, C 0.000 }
gfCNCPoint4[10853] = {X 157.0216, Y 6.4947, Z -5.5000, A 0.000, B 0.000, C 0.000 }
gfCNCPoint4[10854] = {X 157.8154, Y 6.2510, Z -5.5000, A 0.000, B 0.000, C 0.000 }
gfCNCPoint4[10855] = {X 158.6412, Y 6.1637, Z -5.5000, A 0.000, B 0.000, C 0.000 }
gfCNCPoint4[10856] = {X 159.3781, Y 6.1639, Z -5.5000, A 0.000, B 0.000, C 0.000 }
gfCNCPoint4[10857] = {X 160.3301, Y 6.2828, Z -5.5000, A 0.000, B 0.000, C 0.000 }
gfCNCPoint4[10858] = {X 161.2324, Y 6.6088, Z -5.5000, A 0.000, B 0.000, C 0.000 }
gfCNCPoint4[10859] = {X 162.0405, Y 7.1260, Z -5.5000, A 0.000, B 0.000, C 0.000 }
gfCNCPoint4[10860] = {X 162.7145, Y 7.8088, Z -5.5000, A 0.000, B 0.000, C 0.000 }
gfCNCPoint4[10861] = {X 163.2212, Y 8.6236, Z -5.5000, A 0.000, B 0.000, C 0.000 }
gfCNCPoint4[10862] = {X 163.5355, Y 9.5300, Z -5.5000, A 0.000, B 0.000, C 0.000 }
gfCNCPoint4[10863] = {X 163.6421, Y 10.4835, Z -5.5000, A 0.000, B 0.000, C 0.000 }
gfCNCPoint4[10864] = {X 163.6421, Y 17.4615, Z -5.5000, A 0.000, B 0.000, C 0.000 }
gfCNCPoint4[10865] = {X 163.5355, Y 18.4152, Z -5.5000, A 0.000, B 0.000, C 0.000 }
gfCNCPoint4[10866] = {X 163.2211, Y 19.3218, Z -5.5000, A 0.000, B 0.000, C 0.000 }
gfCNCPoint4[10867] = {X 162.7142, Y 20.1366, Z -5.5000, A 0.000, B 0.000, C 0.000 }
gfCNCPoint4[10868] = {X 162.0400, Y 20.8194, Z -5.5000, A 0.000, B 0.000, C 0.000 }
gfCNCPoint4[10869] = {X 161.2318, Y 21.3365, Z -5.5000, A 0.000, B 0.000, C 0.000 }
gfCNCPoint4[10870] = {X 160.3292, Y 21.6625, Z -5.5000, A 0.000, B 0.000, C 0.000 }
gfCNCPoint4[10871] = {X 159.3770, Y 21.7812, Z -5.5000, A 0.000, B 0.000, C 0.000 }
gfCNCPoint4[10872] = {X 158.6793, Y 21.7815, Z -5.5000, A 0.000, B 0.000, C 0.000 }
gfCNCPoint4[10873] = {X 157.8409, Y 21.6967, Z -5.5000, A 0.000, B 0.000, C 0.000 }
gfCNCPoint4[10874] = {X 157.0346, Y 21.4519, Z -5.5000, A 0.000, B 0.000, C 0.000 }
gfCNCPoint4[10875] = {X 156.2905, Y 21.0563, Z -5.5000, A 0.000, B 0.000, C 0.000 }
gfCNCPoint4[10876] = {X 155.6366, Y 20.5248, Z -5.5000, A 0.000, B 0.000, C 0.000 }
gfCNCPoint4[10877] = {X 155.0974, Y 19.8773, Z -5.5000, A 0.000, B 0.000, C 0.000 }
gfCNCPoint4[10878] = {X 152.2767, Y 19.8784, Z -5.5000, A 0.000, B 0.000, C 0.000 }
gfCNCPoint4[10879] = {X 152.2754, Y 40.8742, Z -5.5000, A 0.000, B 0.000, C 0.000 }
gfCNCPoint4[10880] = {X 152.7408, Y 41.3753, Z -5.5000, A 0.000, B 0.000, C 0.000 }
gfCNCPoint4[10881] = {X 152.8361, Y 41.4888, Z -5.5000, A 0.000, B 0.000, C 0.000 }
gfCNCPoint4[10882] = {X 153.3617, Y 42.3141, Z -5.5000, A 0.000, B 0.000, C 0.000 }
gfCNCPoint4[10883] = {X 153.6895, Y 43.2359, Z -5.5000, A 0.000, B 0.000, C 0.000 }
gfCNCPoint4[10884] = {X 153.8031, Y 44.2077, Z -5.5000, A 0.000, B 0.000, C 0.000 }
gfCNCPoint4[10885] = {X 153.8029, Y 45.0415, Z -5.5000, A 0.000, B 0.000, C 0.000 }
gfCNCPoint4[10886] = {X 153.6867, Y 45.9960, Z -5.5000, A 0.000, B 0.000, C 0.000 }
gfCNCPoint4[10887] = {X 153.3623, Y 46.9011, Z -5.5000, A 0.000, B 0.000, C 0.000 }
gfCNCPoint4[10888] = {X 152.8458, Y 47.7120, Z -5.5000, A 0.000, B 0.000, C 0.000 }
gfCNCPoint4[10889] = {X 152.1626, Y 48.3886, Z -5.5000, A 0.000, B 0.000, C 0.000 }
gfCNCPoint4[10890] = {X 151.3468, Y 48.8973, Z -5.5000, A 0.000, B 0.000, C 0.000 }
gfCNCPoint4[10891] = {X 150.4386, Y 49.2130, Z -5.5000, A 0.000, B 0.000, C 0.000 }
